LIN {X 0,Y 523.923,Z 138.219,A -85,B 0,C 180,E1 -4837.939,E2 -4837.939} C_VEL
LIN {X 0,Y 523.904,Z 138.224,A -85,B 0,C 180,E1 -4840.405,E2 -4840.405} C_VEL
LIN {X 0,Y 523.904,Z 138.223,A -85,B 0,C 180,E1 -4842.835,E2 -4842.835} C_VEL
LIN {X 0,Y 523.924,Z 138.217,A -85,B 0,C 180,E1 -4845.234,E2 -4845.234} C_VEL
LIN {X 0,Y 523.964,Z 138.218,A -85,B 0,C 180,E1 -4848.393,E2 -4848.393} C_VEL
LIN {X 0,Y 523.949,Z 138.215,A -85,B 0,C 180,E1 -4851.515,E2 -4851.515} C_VEL
LIN {X 0,Y 524.03,Z 138.208,A -85,B 0,C 180,E1 -4854.613,E2 -4854.613} C_VEL
LIN {X 0,Y 524.106,Z 138.195,A -85,B 0,C 180,E1 -4857.694,E2 -4857.694} C_VEL
LIN {X 0,Y 524.1,Z 138.202,A -85,B 0,C 180,E1 -4860,E2 -4860} C_VEL
LIN {X 0,Y 524.107,Z 138.201,A -85,B 0,C 180,E1 -4862.306,E2 -4862.306} C_VEL
LIN {X 0,Y 524.004,Z 138.215,A -85,B 0,C 180,E1 -4866.16,E2 -4866.16} C_VEL
LIN {X 0,Y 523.948,Z 138.215,A -85,B 0,C 180,E1 -4869.263,E2 -4869.263} C_VEL
LIN {X 0,Y 523.949,Z 138.217,A -85,B 0,C 180,E1 -4872.393,E2 -4872.393} C_VEL
LIN {X 0,Y 523.916,Z 138.224,A -85,B 0,C 180,E1 -4875.562,E2 -4875.562} C_VEL
LIN {X 0,Y 523.916,Z 138.219,A -85,B 0,C 180,E1 -4878.781,E2 -4878.781} C_VEL
LIN {X 0,Y 523.907,Z 138.222,A -85,B 0,C 180,E1 -4881.235,E2 -4881.235} C_VEL
LIN {X 0,Y 523.936,Z 138.22,A -85,B 0,C 180,E1 -4884.196,E2 -4884.196} C_VEL
LIN {X 0,Y 523.9,Z 138.226,A -85,B 0,C 180,E1 -4887.136,E2 -4887.136} C_VEL
LIN {X 0,Y 523.886,Z 138.23,A -85,B 0,C 180,E1 -4889.76,E2 -4889.76} C_VEL
LIN {X 0,Y 523.934,Z 138.219,A -85,B 0,C 180,E1 -4892.45,E2 -4892.45} C_VEL
LIN {X 0,Y 523.917,Z 138.226,A -85,B 0,C 180,E1 -4895.227,E2 -4895.227} C_VEL
LIN {X 0,Y 523.991,Z 138.296,A -85,B 0,C 180,E1 -4897.62,E2 -4897.62} C_VEL
LIN {X 0,Y 524.607,Z 144.392,A -85,B 0,C 180,E1 -4898.768,E2 -4898.768} C_VEL
LIN {X 0,Y 524.385,Z 160.445,A -85,B 0,C 180,E1 -4901.685,E2 -4901.685} C_VEL
LIN {X 0,Y 524.325,Z 167.357,A -85,B 0,C 180,E1 -4902.909,E2 -4902.909} C_VEL
LIN {X 0,Y 525.972,Z 176.481,A -85,B 0,C 180,E1 -4903.087,E2 -4903.087} C_VEL
LIN {X 0,Y 525.921,Z 195.473,A -85,B 0,C 180,E1 -4903.35,E2 -4903.35} C_VEL
LIN {X 0,Y 525.202,Z 201.318,A -85,B 0,C 180,E1 -4903.41,E2 -4903.41} C_VEL
LIN {X 0,Y 519.539,Z 220.31,A -85,B 0,C 180,E1 -4903.516,E2 -4903.516} C_VEL
LIN {X 0,Y 518.88,Z 226.152,A -85,B 0,C 180,E1 -4903.58,E2 -4903.58} C_VEL
LIN {X 0,Y 518.615,Z 274.692,A -85,B 0,C 180,E1 -4904.279,E2 -4904.279} C_VEL
LIN {X 0,Y 518.446,Z 287.858,A -85,B 0,C 180,E1 -4904.627,E2 -4904.627} C_VEL
LIN {X 0,Y 518.237,Z 299.345,A -85,B 0,C 180,E1 -4905.071,E2 -4905.071} C_VEL
LIN {X 0,Y 517.963,Z 309.998,A -85,B 0,C 180,E1 -4905.614,E2 -4905.614} C_VEL
LIN {X 0,Y 517.659,Z 320.815,A -85,B 0,C 180,E1 -4906.314,E2 -4906.314} C_VEL
LIN {X 0,Y 517.334,Z 331.814,A -85,B 0,C 180,E1 -4907.214,E2 -4907.214} C_VEL
LIN {X 0,Y 517.079,Z 341.89,A -85,B 0,C 180,E1 -4908.241,E2 -4908.241} C_VEL
LIN {X 0,Y 516.84,Z 349.994,A -85,B 0,C 180,E1 -4909.254,E2 -4909.254} C_VEL
LIN {X 0,Y 516.698,Z 356.638,A -85,B 0,C 180,E1 -4910.261,E2 -4910.261} C_VEL
LIN {X 0,Y 516.521,Z 363.204,A -85,B 0,C 180,E1 -4911.487,E2 -4911.487} C_VEL
LIN {X 0,Y 516.4,Z 368.418,A -85,B 0,C 180,E1 -4912.726,E2 -4912.726} C_VEL
LIN {X 0,Y 516.269,Z 372.957,A -85,B 0,C 180,E1 -4914.171,E2 -4914.171} C_VEL
LIN {X 0,Y 516.228,Z 375.099,A -85,B 0,C 180,E1 -4915.124,E2 -4915.124} C_VEL
LIN {X 0,Y 516.183,Z 376.74,A -85,B 0,C 180,E1 -4916.154,E2 -4916.154} C_VEL
LIN {X 0,Y 516.182,Z 377.808,A -85,B 0,C 180,E1 -4917.582,E2 -4917.582} C_VEL
LIN {X 0,Y 516.208,Z 377.531,A -85,B 0,C 180,E1 -4919.062,E2 -4919.062} C_VEL
LIN {X 0,Y 516.245,Z 375.742,A -85,B 0,C 180,E1 -4920.608,E2 -4920.608} C_VEL
LIN {X 0,Y 516.255,Z 373.847,A -85,B 0,C 180,E1 -4921.545,E2 -4921.545} C_VEL
LIN {X 0,Y 516.352,Z 370.125,A -85,B 0,C 180,E1 -4922.873,E2 -4922.873} C_VEL
LIN {X 0,Y 516.487,Z 365.084,A -85,B 0,C 180,E1 -4924.187,E2 -4924.187} C_VEL
LIN {X 0,Y 516.59,Z 358.966,A -85,B 0,C 180,E1 -4925.416,E2 -4925.416} C_VEL
LIN {X 0,Y 516.767,Z 351.875,A -85,B 0,C 180,E1 -4926.559,E2 -4926.559} C_VEL
LIN {X 0,Y 517,Z 343.744,A -85,B 0,C 180,E1 -4927.627,E2 -4927.627} C_VEL
LIN {X 0,Y 517.281,Z 333.786,A -85,B 0,C 180,E1 -4928.688,E2 -4928.688} C_VEL
LIN {X 0,Y 517.613,Z 322.557,A -85,B 0,C 180,E1 -4929.639,E2 -4929.639} C_VEL
LIN {X 0,Y 517.953,Z 311.621,A -85,B 0,C 180,E1 -4930.377,E2 -4930.377} C_VEL
LIN {X 0,Y 518.172,Z 299.685,A -85,B 0,C 180,E1 -4931.003,E2 -4931.003} C_VEL
LIN {X 0,Y 518.477,Z 286.399,A -85,B 0,C 180,E1 -4931.509,E2 -4931.509} C_VEL
LIN {X 0,Y 518.628,Z 274.047,A -85,B 0,C 180,E1 -4931.824,E2 -4931.824} C_VEL
LIN {X 0,Y 519.033,Z 177.008,A -85,B 0,C 180,E1 -4933.201,E2 -4933.201} C_VEL
LIN {X 0,Y 517.288,Z 167.26,A -85,B 0,C 180,E1 -4933.397,E2 -4933.397} C_VEL
LIN {X 0,Y 517.567,Z 152.131,A -85,B 0,C 180,E1 -4936.253,E2 -4936.253} C_VEL
LIN {X 0,Y 517.652,Z 143.863,A -85,B 0,C 180,E1 -4937.83,E2 -4937.83} C_VEL
LIN {X 0,Y 516.982,Z 139.092,A -85,B 0,C 180,E1 -4938.78,E2 -4938.78} C_VEL
LIN {X 0,Y 516.956,Z 139.089,A -85,B 0,C 180,E1 -4941.399,E2 -4941.399} C_VEL
LIN {X 0,Y 517.014,Z 139.087,A -85,B 0,C 180,E1 -4944.54,E2 -4944.54} C_VEL
LIN {X 0,Y 517.082,Z 139.07,A -85,B 0,C 180,E1 -4947.663,E2 -4947.663} C_VEL
LIN {X 0,Y 517.09,Z 139.072,A -85,B 0,C 180,E1 -4950.779,E2 -4950.779} C_VEL
LIN {X 0,Y 516.949,Z 139.087,A -85,B 0,C 180,E1 -4953.117,E2 -4953.117} C_VEL
LIN {X 0,Y 516.975,Z 139.092,A -85,B 0,C 180,E1 -4956.244,E2 -4956.244} C_VEL
LIN {X 0,Y 516.94,Z 139.088,A -85,B 0,C 180,E1 -4959.39,E2 -4959.39} C_VEL
LIN {X 0,Y 516.956,Z 139.09,A -85,B 0,C 180,E1 -4961.807,E2 -4961.807} C_VEL
LIN {X 0,Y 516.942,Z 139.088,A -85,B 0,C 180,E1 -4965.144,E2 -4965.144} C_VEL
LIN {X 0,Y 516.878,Z 139.1,A -85,B 0,C 180,E1 -4968.224,E2 -4968.224} C_VEL
LIN {X 0,Y 516.902,Z 139.093,A -85,B 0,C 180,E1 -4970.702,E2 -4970.702} C_VEL
LIN {X 0,Y 516.859,Z 139.099,A -85,B 0,C 180,E1 -4973.224,E2 -4973.224} C_VEL
LIN {X 0,Y 516.884,Z 139.098,A -85,B 0,C 180,E1 -4976.182,E2 -4976.182} C_VEL
LIN {X 0,Y 516.906,Z 139.096,A -85,B 0,C 180,E1 -4979.306,E2 -4979.306} C_VEL
LIN {X 0,Y 516.897,Z 139.093,A -85,B 0,C 180,E1 -4982.543,E2 -4982.543} C_VEL
LIN {X 0,Y 516.863,Z 139.103,A -85,B 0,C 180,E1 -4985.329,E2 -4985.329} C_VEL
LIN {X 0,Y 516.88,Z 139.098,A -85,B 0,C 180,E1 -4987.943,E2 -4987.943} C_VEL
LIN {X 0,Y 516.856,Z 139.099,A -85,B 0,C 180,E1 -4990.745,E2 -4990.745} C_VEL
LIN {X 0,Y 516.883,Z 139.096,A -85,B 0,C 180,E1 -4993.904,E2 -4993.904} C_VEL
LIN {X 0,Y 516.883,Z 139.095,A -85,B 0,C 180,E1 -4996.107,E2 -4996.107} C_VEL
LIN {X 0,Y 516.856,Z 139.106,A -85,B 0,C 180,E1 -4999.255,E2 -4999.255} C_VEL
LIN {X 0,Y 516.863,Z 139.097,A -85,B 0,C 180,E1 -5002.274,E2 -5002.274} C_VEL
LIN {X 0,Y 516.876,Z 139.103,A -85,B 0,C 180,E1 -5005.174,E2 -5005.174} C_VEL
LIN {X 0,Y 516.869,Z 139.096,A -85,B 0,C 180,E1 -5007.975,E2 -5007.975} C_VEL
LIN {X 0,Y 516.902,Z 139.098,A -85,B 0,C 180,E1 -5010.694,E2 -5010.694} C_VEL
LIN {X 0,Y 516.885,Z 139.094,A -85,B 0,C 180,E1 -5013.818,E2 -5013.818} C_VEL
LIN {X 0,Y 516.847,Z 139.108,A -85,B 0,C 180,E1 -5016.775,E2 -5016.775} C_VEL
LIN {X 0,Y 516.911,Z 139.091,A -85,B 0,C 180,E1 -5019.742,E2 -5019.742} C_VEL
LIN {X 0,Y 516.869,Z 139.105,A -85,B 0,C 180,E1 -5022.594,E2 -5022.594} C_VEL
LIN {X 0,Y 516.935,Z 139.091,A -85,B 0,C 180,E1 -5025.03,E2 -5025.03} C_VEL
LIN {X 0,Y 516.972,Z 139.089,A -85,B 0,C 180,E1 -5028.234,E2 -5028.234} C_VEL
LIN {X 0,Y 516.925,Z 139.09,A -85,B 0,C 180,E1 -5031.399,E2 -5031.399} C_VEL
LIN {X 0,Y 516.984,Z 139.088,A -85,B 0,C 180,E1 -5034.539,E2 -5034.539} C_VEL
LIN {X 0,Y 517.076,Z 139.072,A -85,B 0,C 180,E1 -5037.663,E2 -5037.663} C_VEL
LIN {X 0,Y 517.069,Z 139.078,A -85,B 0,C 180,E1 -5040,E2 -5040} C_VEL
LIN {X 0,Y 517.076,Z 139.077,A -85,B 0,C 180,E1 -5042.337,E2 -5042.337} C_VEL
LIN {X 0,Y 516.971,Z 139.09,A -85,B 0,C 180,E1 -5046.244,E2 -5046.244} C_VEL
LIN {X 0,Y 516.91,Z 139.093,A -85,B 0,C 180,E1 -5049.39,E2 -5049.39} C_VEL
LIN {X 0,Y 516.89,Z 139.095,A -85,B 0,C 180,E1 -5052.565,E2 -5052.565} C_VEL
LIN {X 0,Y 516.888,Z 139.095,A -85,B 0,C 180,E1 -5055.121,E2 -5055.121} C_VEL
LIN {X 0,Y 516.85,Z 139.101,A -85,B 0,C 180,E1 -5058.225,E2 -5058.225} C_VEL
LIN {X 0,Y 516.866,Z 139.097,A -85,B 0,C 180,E1 -5060.703,E2 -5060.703} C_VEL
LIN {X 0,Y 516.843,Z 139.103,A -85,B 0,C 180,E1 -5063.225,E2 -5063.225} C_VEL
LIN {X 0,Y 516.864,Z 139.098,A -85,B 0,C 180,E1 -5066.177,E2 -5066.177} C_VEL
LIN {X 0,Y 516.832,Z 139.101,A -85,B 0,C 180,E1 -5068.421,E2 -5068.421} C_VEL
LIN {X 0,Y 516.851,Z 139.103,A -85,B 0,C 180,E1 -5071.112,E2 -5071.112} C_VEL
LIN {X 0,Y 516.871,Z 139.098,A -85,B 0,C 180,E1 -5073.959,E2 -5073.959} C_VEL
LIN {X 0,Y 516.809,Z 139.106,A -85,B 0,C 180,E1 -5076.752,E2 -5076.752} C_VEL
LIN {X 0,Y 516.856,Z 139.1,A -85,B 0,C 180,E1 -5079.724,E2 -5079.724} C_VEL
LIN {X 0,Y 516.843,Z 139.104,A -85,B 0,C 180,E1 -5082.836,E2 -5082.836} C_VEL
LIN {X 0,Y 516.898,Z 139.101,A -85,B 0,C 180,E1 -5085.007,E2 -5085.007} C_VEL
LIN {X 0,Y 516.849,Z 139.1,A -85,B 0,C 180,E1 -5088.407,E2 -5088.407} C_VEL
LIN {X 0,Y 516.861,Z 139.102,A -85,B 0,C 180,E1 -5091.282,E2 -5091.282} C_VEL
LIN {X 0,Y 516.828,Z 139.108,A -85,B 0,C 180,E1 -5094.677,E2 -5094.677} C_VEL
LIN {X 0,Y 516.865,Z 139.098,A -85,B 0,C 180,E1 -5097.462,E2 -5097.462} C_VEL
LIN {X 0,Y 516.839,Z 139.108,A -85,B 0,C 180,E1 -5100.491,E2 -5100.491} C_VEL
LIN {X 0,Y 516.83,Z 139.106,A -85,B 0,C 180,E1 -5103.337,E2 -5103.337} C_VEL
LIN {X 0,Y 516.882,Z 139.297,A -85,B 0,C 180,E1 -5105.735,E2 -5105.735} C_VEL
LIN {X 0,Y 518.332,Z 147.82,A -85,B 0,C 180,E1 -5107.221,E2 -5107.221} C_VEL
LIN {X 0,Y 517.928,Z 164.685,A -85,B 0,C 180,E1 -5109.978,E2 -5109.978} C_VEL
LIN {X 0,Y 517.496,Z 182.348,A -85,B 0,C 180,E1 -5112.819,E2 -5112.819} C_VEL
LIN {X 0,Y 517.24,Z 193.77,A -85,B 0,C 180,E1 -5114.636,E2 -5114.636} C_VEL
LIN {X 0,Y 519.026,Z 206.371,A -85,B 0,C 180,E1 -5114.868,E2 -5114.868} C_VEL
LIN {X 0,Y 518.573,Z 302.296,A -85,B 0,C 180,E1 -5116.23,E2 -5116.23} C_VEL
LIN {X 0,Y 518.333,Z 316.173,A -85,B 0,C 180,E1 -5116.598,E2 -5116.598} C_VEL
LIN {X 0,Y 518.051,Z 329.122,A -85,B 0,C 180,E1 -5117.115,E2 -5117.115} C_VEL
LIN {X 0,Y 517.733,Z 341.445,A -85,B 0,C 180,E1 -5117.788,E2 -5117.788} C_VEL
LIN {X 0,Y 517.469,Z 352.266,A -85,B 0,C 180,E1 -5118.543,E2 -5118.543} C_VEL
LIN {X 0,Y 517.166,Z 362.51,A -85,B 0,C 180,E1 -5119.429,E2 -5119.429} C_VEL
LIN {X 0,Y 516.902,Z 371.715,A -85,B 0,C 180,E1 -5120.412,E2 -5120.412} C_VEL
LIN {X 0,Y 516.652,Z 380.678,A -85,B 0,C 180,E1 -5121.591,E2 -5121.591} C_VEL
LIN {X 0,Y 516.502,Z 387.894,A -85,B 0,C 180,E1 -5122.769,E2 -5122.769} C_VEL
LIN {X 0,Y 516.404,Z 394.464,A -85,B 0,C 180,E1 -5124.142,E2 -5124.142} C_VEL
LIN {X 0,Y 516.267,Z 398.806,A -85,B 0,C 180,E1 -5125.315,E2 -5125.315} C_VEL
LIN {X 0,Y 516.352,Z 401.108,A -85,B 0,C 180,E1 -5126.098,E2 -5126.098} C_VEL
LIN {X 0,Y 516.282,Z 402.97,A -85,B 0,C 180,E1 -5126.879,E2 -5126.879} C_VEL
LIN {X 0,Y 516.261,Z 404.367,A -85,B 0,C 180,E1 -5127.659,E2 -5127.659} C_VEL
LIN {X 0,Y 516.162,Z 405.968,A -85,B 0,C 180,E1 -5129.22,E2 -5129.22} C_VEL
LIN {X 0,Y 516.159,Z 406.183,A -85,B 0,C 180,E1 -5130,E2 -5130} C_VEL
LIN {X 0,Y 516.192,Z 405.356,A -85,B 0,C 180,E1 -5131.56,E2 -5131.56} C_VEL
LIN {X 0,Y 516.261,Z 404.358,A -85,B 0,C 180,E1 -5132.341,E2 -5132.341} C_VEL
LIN {X 0,Y 516.282,Z 402.958,A -85,B 0,C 180,E1 -5133.121,E2 -5133.121} C_VEL
LIN {X 0,Y 516.31,Z 400.014,A -85,B 0,C 180,E1 -5134.294,E2 -5134.294} C_VEL
LIN {X 0,Y 516.368,Z 396.03,A -85,B 0,C 180,E1 -5135.467,E2 -5135.467} C_VEL
LIN {X 0,Y 516.441,Z 390.135,A -85,B 0,C 180,E1 -5136.793,E2 -5136.793} C_VEL
LIN {X 0,Y 516.586,Z 383.2,A -85,B 0,C 180,E1 -5138.016,E2 -5138.016} C_VEL
LIN {X 0,Y 516.801,Z 374.888,A -85,B 0,C 180,E1 -5139.195,E2 -5139.195} C_VEL
LIN {X 0,Y 517.005,Z 366.359,A -85,B 0,C 180,E1 -5140.179,E2 -5140.179} C_VEL
LIN {X 0,Y 517.337,Z 355.824,A -85,B 0,C 180,E1 -5141.162,E2 -5141.162} C_VEL
LIN {X 0,Y 517.648,Z 344.821,A -85,B 0,C 180,E1 -5141.989,E2 -5141.989} C_VEL
LIN {X 0,Y 517.935,Z 333.952,A -85,B 0,C 180,E1 -5142.639,E2 -5142.639} C_VEL
LIN {X 0,Y 518.204,Z 322.146,A -85,B 0,C 180,E1 -5143.18,E2 -5143.18} C_VEL
LIN {X 0,Y 518.486,Z 308.535,A -85,B 0,C 180,E1 -5143.622,E2 -5143.622} C_VEL
LIN {X 0,Y 518.664,Z 296.421,A -85,B 0,C 180,E1 -5143.867,E2 -5143.867} C_VEL
LIN {X 0,Y 518.974,Z 204.763,A -85,B 0,C 180,E1 -5145.154,E2 -5145.154} C_VEL
LIN {X 0,Y 517.226,Z 193.408,A -85,B 0,C 180,E1 -5145.389,E2 -5145.389} C_VEL
LIN {X 0,Y 517.683,Z 174.421,A -85,B 0,C 180,E1 -5148.4,E2 -5148.4} C_VEL
LIN {X 0,Y 518.12,Z 155.212,A -85,B 0,C 180,E1 -5151.484,E2 -5151.484} C_VEL
LIN {X 0,Y 518.214,Z 146.498,A -85,B 0,C 180,E1 -5152.904,E2 -5152.904} C_VEL
LIN {X 0,Y 516.884,Z 139.1,A -85,B 0,C 180,E1 -5154.217,E2 -5154.217} C_VEL
LIN {X 0,Y 516.868,Z 139.106,A -85,B 0,C 180,E1 -5157.536,E2 -5157.536} C_VEL
LIN {X 0,Y 516.837,Z 139.104,A -85,B 0,C 180,E1 -5160.208,E2 -5160.208} C_VEL
LIN {X 0,Y 516.86,Z 139.106,A -85,B 0,C 180,E1 -5162.95,E2 -5162.95} C_VEL
LIN {X 0,Y 516.803,Z 139.107,A -85,B 0,C 180,E1 -5165.786,E2 -5165.786} C_VEL
LIN {X 0,Y 516.854,Z 139.103,A -85,B 0,C 180,E1 -5168.719,E2 -5168.719} C_VEL
LIN {X 0,Y 516.832,Z 139.103,A -85,B 0,C 180,E1 -5171.784,E2 -5171.784} C_VEL
LIN {X 0,Y 516.899,Z 139.101,A -85,B 0,C 180,E1 -5175.007,E2 -5175.007} C_VEL
LIN {X 0,Y 516.832,Z 139.104,A -85,B 0,C 180,E1 -5178.41,E2 -5178.41} C_VEL
LIN {X 0,Y 516.856,Z 139.103,A -85,B 0,C 180,E1 -5181.282,E2 -5181.282} C_VEL
LIN {X 0,Y 516.827,Z 139.108,A -85,B 0,C 180,E1 -5184.677,E2 -5184.677} C_VEL
LIN {X 0,Y 516.866,Z 139.097,A -85,B 0,C 180,E1 -5187.463,E2 -5187.463} C_VEL
LIN {X 0,Y 516.841,Z 139.105,A -85,B 0,C 180,E1 -5190.491,E2 -5190.491} C_VEL
LIN {X 0,Y 516.831,Z 139.102,A -85,B 0,C 180,E1 -5193.337,E2 -5193.337} C_VEL
LIN {X 0,Y 516.861,Z 139.096,A -85,B 0,C 180,E1 -5195.925,E2 -5195.925} C_VEL
LIN {X 0,Y 516.853,Z 139.106,A -85,B 0,C 180,E1 -5198.461,E2 -5198.461} C_VEL
LIN {X 0,Y 516.849,Z 139.103,A -85,B 0,C 180,E1 -5200.953,E2 -5200.953} C_VEL
LIN {X 0,Y 516.836,Z 139.099,A -85,B 0,C 180,E1 -5203.408,E2 -5203.408} C_VEL
LIN {X 0,Y 516.852,Z 139.1,A -85,B 0,C 180,E1 -5205.832,E2 -5205.832} C_VEL
LIN {X 0,Y 516.924,Z 139.096,A -85,B 0,C 180,E1 -5208.233,E2 -5208.233} C_VEL
LIN {X 0,Y 516.923,Z 139.09,A -85,B 0,C 180,E1 -5211.399,E2 -5211.399} C_VEL
LIN {X 0,Y 516.981,Z 139.087,A -85,B 0,C 180,E1 -5214.539,E2 -5214.539} C_VEL
LIN {X 0,Y 517.075,Z 139.071,A -85,B 0,C 180,E1 -5217.663,E2 -5217.663} C_VEL
LIN {X 0,Y 517.069,Z 139.078,A -85,B 0,C 180,E1 -5220,E2 -5220} C_VEL
LIN {X 0,Y 517.076,Z 139.076,A -85,B 0,C 180,E1 -5222.337,E2 -5222.337} C_VEL
LIN {X 0,Y 516.971,Z 139.09,A -85,B 0,C 180,E1 -5226.244,E2 -5226.244} C_VEL
LIN {X 0,Y 516.91,Z 139.092,A -85,B 0,C 180,E1 -5229.39,E2 -5229.39} C_VEL
LIN {X 0,Y 516.902,Z 139.093,A -85,B 0,C 180,E1 -5232.565,E2 -5232.565} C_VEL
LIN {X 0,Y 516.941,Z 139.089,A -85,B 0,C 180,E1 -5235.142,E2 -5235.142} C_VEL
LIN {X 0,Y 516.873,Z 139.1,A -85,B 0,C 180,E1 -5238.224,E2 -5238.224} C_VEL
LIN {X 0,Y 516.875,Z 139.096,A -85,B 0,C 180,E1 -5240.703,E2 -5240.703} C_VEL
LIN {X 0,Y 516.846,Z 139.103,A -85,B 0,C 180,E1 -5243.225,E2 -5243.225} C_VEL
LIN {X 0,Y 516.883,Z 139.099,A -85,B 0,C 180,E1 -5246.181,E2 -5246.181} C_VEL
LIN {X 0,Y 516.894,Z 139.101,A -85,B 0,C 180,E1 -5249.306,E2 -5249.306} C_VEL
LIN {X 0,Y 516.896,Z 139.096,A -85,B 0,C 180,E1 -5252.542,E2 -5252.542} C_VEL
LIN {X 0,Y 516.864,Z 139.106,A -85,B 0,C 180,E1 -5255.328,E2 -5255.328} C_VEL
LIN {X 0,Y 516.919,Z 139.106,A -85,B 0,C 180,E1 -5257.475,E2 -5257.475} C_VEL
LIN {X 0,Y 517.609,Z 144.246,A -85,B 0,C 180,E1 -5258.46,E2 -5258.46} C_VEL
LIN {X 0,Y 517.433,Z 158.995,A -85,B 0,C 180,E1 -5261.17,E2 -5261.17} C_VEL
LIN {X 0,Y 517.294,Z 167.36,A -85,B 0,C 180,E1 -5262.696,E2 -5262.696} C_VEL
LIN {X 0,Y 519.147,Z 177.868,A -85,B 0,C 180,E1 -5262.902,E2 -5262.902} C_VEL
LIN {X 0,Y 518.88,Z 226.152,A -85,B 0,C 180,E1 -5263.58,E2 -5263.58} C_VEL
LIN {X 0,Y 518.205,Z 231.997,A -85,B 0,C 180,E1 -5263.643,E2 -5263.643} C_VEL
LIN {X 0,Y 512.511,Z 250.987,A -85,B 0,C 180,E1 -5263.75,E2 -5263.75} C_VEL
LIN {X 0,Y 511.88,Z 256.829,A -85,B 0,C 180,E1 -5263.816,E2 -5263.816} C_VEL
LIN {X 0,Y 511.741,Z 276.642,A -85,B 0,C 180,E1 -5264.132,E2 -5264.132} C_VEL
LIN {X 0,Y 511.526,Z 289.245,A -85,B 0,C 180,E1 -5264.484,E2 -5264.484} C_VEL
LIN {X 0,Y 511.276,Z 301.879,A -85,B 0,C 180,E1 -5265.003,E2 -5265.003} C_VEL
LIN {X 0,Y 510.929,Z 313.813,A -85,B 0,C 180,E1 -5265.666,E2 -5265.666} C_VEL
LIN {X 0,Y 510.649,Z 323.936,A -85,B 0,C 180,E1 -5266.38,E2 -5266.38} C_VEL
LIN {X 0,Y 510.331,Z 334.534,A -85,B 0,C 180,E1 -5267.304,E2 -5267.304} C_VEL
LIN {X 0,Y 510.006,Z 343.981,A -85,B 0,C 180,E1 -5268.331,E2 -5268.331} C_VEL
LIN {X 0,Y 509.768,Z 352.414,A -85,B 0,C 180,E1 -5269.459,E2 -5269.459} C_VEL
LIN {X 0,Y 509.529,Z 359.455,A -85,B 0,C 180,E1 -5270.618,E2 -5270.618} C_VEL
LIN {X 0,Y 509.381,Z 365.472,A -85,B 0,C 180,E1 -5271.854,E2 -5271.854} C_VEL
LIN {X 0,Y 509.303,Z 370.387,A -85,B 0,C 180,E1 -5273.164,E2 -5273.164} C_VEL
LIN {X 0,Y 509.141,Z 374.221,A -85,B 0,C 180,E1 -5274.566,E2 -5274.566} C_VEL
LIN {X 0,Y 509.086,Z 376.655,A -85,B 0,C 180,E1 -5275.926,E2 -5275.926} C_VEL
LIN {X 0,Y 509.093,Z 377.969,A -85,B 0,C 180,E1 -5277.425,E2 -5277.425} C_VEL
LIN {X 0,Y 509.118,Z 377.859,A -85,B 0,C 180,E1 -5278.856,E2 -5278.856} C_VEL
LIN {X 0,Y 509.132,Z 376.278,A -85,B 0,C 180,E1 -5280.418,E2 -5280.418} C_VEL
LIN {X 0,Y 509.185,Z 374.104,A -85,B 0,C 180,E1 -5281.563,E2 -5281.563} C_VEL
LIN {X 0,Y 509.273,Z 370.409,A -85,B 0,C 180,E1 -5282.909,E2 -5282.909} C_VEL
LIN {X 0,Y 509.426,Z 365.403,A -85,B 0,C 180,E1 -5284.242,E2 -5284.242} C_VEL
LIN {X 0,Y 509.557,Z 358.926,A -85,B 0,C 180,E1 -5285.558,E2 -5285.558} C_VEL
LIN {X 0,Y 509.756,Z 350.795,A -85,B 0,C 180,E1 -5286.863,E2 -5286.863} C_VEL
LIN {X 0,Y 510.022,Z 342.281,A -85,B 0,C 180,E1 -5287.955,E2 -5287.955} C_VEL
LIN {X 0,Y 510.363,Z 331.972,A -85,B 0,C 180,E1 -5289.02,E2 -5289.02} C_VEL
LIN {X 0,Y 510.672,Z 321.732,A -85,B 0,C 180,E1 -5289.876,E2 -5289.876} C_VEL
LIN {X 0,Y 511.075,Z 310.445,A -85,B 0,C 180,E1 -5290.625,E2 -5290.625} C_VEL
LIN {X 0,Y 511.3,Z 297.836,A -85,B 0,C 180,E1 -5291.269,E2 -5291.269} C_VEL
LIN {X 0,Y 511.575,Z 285.248,A -85,B 0,C 180,E1 -5291.736,E2 -5291.736} C_VEL
LIN {X 0,Y 511.765,Z 271.826,A -85,B 0,C 180,E1 -5292.053,E2 -5292.053} C_VEL
LIN {X 0,Y 512.157,Z 177.465,A -85,B 0,C 180,E1 -5293.405,E2 -5293.405} C_VEL
LIN {X 0,Y 510.291,Z 167.361,A -85,B 0,C 180,E1 -5293.626,E2 -5293.626} C_VEL
LIN {X 0,Y 510.646,Z 151.393,A -85,B 0,C 180,E1 -5296.672,E2 -5296.672} C_VEL
LIN {X 0,Y 510.609,Z 144.09,A -85,B 0,C 180,E1 -5298.085,E2 -5298.085} C_VEL
LIN {X 0,Y 509.94,Z 139.968,A -85,B 0,C 180,E1 -5298.925,E2 -5298.925} C_VEL
LIN {X 0,Y 509.911,Z 139.969,A -85,B 0,C 180,E1 -5302.078,E2 -5302.078} C_VEL
LIN {X 0,Y 509.965,Z 139.965,A -85,B 0,C 180,E1 -5304.464,E2 -5304.464} C_VEL
LIN {X 0,Y 510.052,Z 139.946,A -85,B 0,C 180,E1 -5307.631,E2 -5307.631} C_VEL
LIN {X 0,Y 510.04,Z 139.95,A -85,B 0,C 180,E1 -5310.79,E2 -5310.79} C_VEL
LIN {X 0,Y 510.047,Z 139.955,A -85,B 0,C 180,E1 -5312.369,E2 -5312.369} C_VEL
LIN {X 0,Y 509.945,Z 139.96,A -85,B 0,C 180,E1 -5315.536,E2 -5315.536} C_VEL
LIN {X 0,Y 509.891,Z 139.968,A -85,B 0,C 180,E1 -5318.721,E2 -5318.721} C_VEL
LIN {X 0,Y 509.908,Z 139.97,A -85,B 0,C 180,E1 -5321.932,E2 -5321.932} C_VEL
LIN {X 0,Y 509.898,Z 139.965,A -85,B 0,C 180,E1 -5325.242,E2 -5325.242} C_VEL
LIN {X 0,Y 509.837,Z 139.974,A -85,B 0,C 180,E1 -5328.485,E2 -5328.485} C_VEL
LIN {X 0,Y 509.845,Z 139.972,A -85,B 0,C 180,E1 -5331.002,E2 -5331.002} C_VEL
LIN {X 0,Y 509.821,Z 139.98,A -85,B 0,C 180,E1 -5333.564,E2 -5333.564} C_VEL
LIN {X 0,Y 509.821,Z 139.976,A -85,B 0,C 180,E1 -5336.357,E2 -5336.357} C_VEL
LIN {X 0,Y 509.839,Z 139.972,A -85,B 0,C 180,E1 -5338.847,E2 -5338.847} C_VEL
LIN {X 0,Y 509.822,Z 139.983,A -85,B 0,C 180,E1 -5341.59,E2 -5341.59} C_VEL
LIN {X 0,Y 509.837,Z 139.973,A -85,B 0,C 180,E1 -5344.415,E2 -5344.415} C_VEL
LIN {X 0,Y 509.81,Z 139.983,A -85,B 0,C 180,E1 -5347.342,E2 -5347.342} C_VEL
LIN {X 0,Y 509.817,Z 139.975,A -85,B 0,C 180,E1 -5350.385,E2 -5350.385} C_VEL
LIN {X 0,Y 509.809,Z 139.981,A -85,B 0,C 180,E1 -5353.573,E2 -5353.573} C_VEL
LIN {X 0,Y 509.808,Z 139.976,A -85,B 0,C 180,E1 -5356.427,E2 -5356.427} C_VEL
LIN {X 0,Y 509.817,Z 139.978,A -85,B 0,C 180,E1 -5359.615,E2 -5359.615} C_VEL
LIN {X 0,Y 509.811,Z 139.979,A -85,B 0,C 180,E1 -5362.658,E2 -5362.658} C_VEL
LIN {X 0,Y 509.843,Z 139.972,A -85,B 0,C 180,E1 -5365.801,E2 -5365.801} C_VEL
LIN {X 0,Y 509.84,Z 139.978,A -85,B 0,C 180,E1 -5368.722,E2 -5368.722} C_VEL
LIN {X 0,Y 509.82,Z 139.975,A -85,B 0,C 180,E1 -5371.917,E2 -5371.917} C_VEL
LIN {X 0,Y 509.805,Z 139.984,A -85,B 0,C 180,E1 -5374.7,E2 -5374.7} C_VEL
LIN {X 0,Y 509.828,Z 139.974,A -85,B 0,C 180,E1 -5377.459,E2 -5377.459} C_VEL
LIN {X 0,Y 509.894,Z 139.966,A -85,B 0,C 180,E1 -5379.844,E2 -5379.844} C_VEL
LIN {X 0,Y 509.851,Z 139.976,A -85,B 0,C 180,E1 -5382.347,E2 -5382.347} C_VEL
LIN {X 0,Y 509.889,Z 139.971,A -85,B 0,C 180,E1 -5384.818,E2 -5384.818} C_VEL
LIN {X 0,Y 509.906,Z 139.968,A -85,B 0,C 180,E1 -5388.124,E2 -5388.124} C_VEL
LIN {X 0,Y 509.878,Z 139.968,A -85,B 0,C 180,E1 -5391.279,E2 -5391.279} C_VEL
LIN {X 0,Y 509.92,Z 139.963,A -85,B 0,C 180,E1 -5393.67,E2 -5393.67} C_VEL
LIN {X 0,Y 509.89,Z 139.968,A -85,B 0,C 180,E1 -5396.839,E2 -5396.839} C_VEL
LIN {X 0,Y 509.928,Z 139.967,A -85,B 0,C 180,E1 -5398.42,E2 -5398.42} C_VEL
LIN {X 0,Y 510.038,Z 139.954,A -85,B 0,C 180,E1 -5400,E2 -5400} C_VEL
LIN {X 0,Y 510.045,Z 139.952,A -85,B 0,C 180,E1 -5402.369,E2 -5402.369} C_VEL
LIN {X 0,Y 509.938,Z 139.962,A -85,B 0,C 180,E1 -5405.536,E2 -5405.536} C_VEL
LIN {X 0,Y 509.879,Z 139.975,A -85,B 0,C 180,E1 -5407.923,E2 -5407.923} C_VEL
LIN {X 0,Y 509.865,Z 139.969,A -85,B 0,C 180,E1 -5411.127,E2 -5411.127} C_VEL
LIN {X 0,Y 509.821,Z 139.979,A -85,B 0,C 180,E1 -5413.553,E2 -5413.553} C_VEL
LIN {X 0,Y 509.794,Z 139.984,A -85,B 0,C 180,E1 -5416.005,E2 -5416.005} C_VEL
LIN {X 0,Y 509.812,Z 139.976,A -85,B 0,C 180,E1 -5418.486,E2 -5418.486} C_VEL
LIN {X 0,Y 509.816,Z 139.976,A -85,B 0,C 180,E1 -5421.003,E2 -5421.003} C_VEL
LIN {X 0,Y 509.805,Z 139.985,A -85,B 0,C 180,E1 -5423.565,E2 -5423.565} C_VEL
LIN {X 0,Y 509.804,Z 139.977,A -85,B 0,C 180,E1 -5426.353,E2 -5426.353} C_VEL
LIN {X 0,Y 509.796,Z 139.979,A -85,B 0,C 180,E1 -5428.849,E2 -5428.849} C_VEL
LIN {X 0,Y 509.791,Z 139.985,A -85,B 0,C 180,E1 -5431.592,E2 -5431.592} C_VEL
LIN {X 0,Y 509.83,Z 139.973,A -85,B 0,C 180,E1 -5434.415,E2 -5434.415} C_VEL
LIN {X 0,Y 509.777,Z 139.988,A -85,B 0,C 180,E1 -5437.344,E2 -5437.344} C_VEL
LIN {X 0,Y 509.814,Z 139.976,A -85,B 0,C 180,E1 -5440.385,E2 -5440.385} C_VEL
LIN {X 0,Y 509.794,Z 139.981,A -85,B 0,C 180,E1 -5443.575,E2 -5443.575} C_VEL
LIN {X 0,Y 509.794,Z 139.979,A -85,B 0,C 180,E1 -5446.425,E2 -5446.425} C_VEL
LIN {X 0,Y 509.796,Z 139.979,A -85,B 0,C 180,E1 -5449.613,E2 -5449.613} C_VEL
LIN {X 0,Y 509.776,Z 139.985,A -85,B 0,C 180,E1 -5452.655,E2 -5452.655} C_VEL
LIN {X 0,Y 509.829,Z 139.973,A -85,B 0,C 180,E1 -5455.802,E2 -5455.802} C_VEL
LIN {X 0,Y 509.816,Z 139.984,A -85,B 0,C 180,E1 -5458.726,E2 -5458.726} C_VEL
LIN {X 0,Y 509.823,Z 139.978,A -85,B 0,C 180,E1 -5462.05,E2 -5462.05} C_VEL
LIN {X 0,Y 509.784,Z 139.988,A -85,B 0,C 180,E1 -5464.699,E2 -5464.699} C_VEL
LIN {X 0,Y 509.828,Z 140.028,A -85,B 0,C 180,E1 -5465.533,E2 -5465.533} C_VEL
LIN {X 0,Y 511.376,Z 148.534,A -85,B 0,C 180,E1 -5467.044,E2 -5467.044} C_VEL
LIN {X 0,Y 511.01,Z 163.696,A -85,B 0,C 180,E1 -5469.561,E2 -5469.561} C_VEL
LIN {X 0,Y 510.592,Z 178.964,A -85,B 0,C 180,E1 -5472.057,E2 -5472.057} C_VEL
LIN {X 0,Y 510.261,Z 193.653,A -85,B 0,C 180,E1 -5474.422,E2 -5474.422} C_VEL
LIN {X 0,Y 512.181,Z 206.085,A -85,B 0,C 180,E1 -5474.66,E2 -5474.66} C_VEL
LIN {X 0,Y 511.69,Z 301.999,A -85,B 0,C 180,E1 -5476.041,E2 -5476.041} C_VEL
LIN {X 0,Y 511.456,Z 315.147,A -85,B 0,C 180,E1 -5476.39,E2 -5476.39} C_VEL
LIN {X 0,Y 511.132,Z 327.819,A -85,B 0,C 180,E1 -5476.887,E2 -5476.887} C_VEL
LIN {X 0,Y 510.823,Z 339.597,A -85,B 0,C 180,E1 -5477.517,E2 -5477.517} C_VEL
LIN {X 0,Y 510.524,Z 350.748,A -85,B 0,C 180,E1 -5478.284,E2 -5478.284} C_VEL
LIN {X 0,Y 510.213,Z 361.239,A -85,B 0,C 180,E1 -5479.183,E2 -5479.183} C_VEL
LIN {X 0,Y 509.898,Z 369.813,A -85,B 0,C 180,E1 -5480.079,E2 -5480.079} C_VEL
LIN {X 0,Y 509.661,Z 377.723,A -85,B 0,C 180,E1 -5481.075,E2 -5481.075} C_VEL
LIN {X 0,Y 509.461,Z 385.449,A -85,B 0,C 180,E1 -5482.27,E2 -5482.27} C_VEL
LIN {X 0,Y 509.308,Z 392.562,A -85,B 0,C 180,E1 -5483.662,E2 -5483.662} C_VEL
LIN {X 0,Y 509.241,Z 397.295,A -85,B 0,C 180,E1 -5484.853,E2 -5484.853} C_VEL
LIN {X 0,Y 509.245,Z 400.912,A -85,B 0,C 180,E1 -5486.043,E2 -5486.043} C_VEL
LIN {X 0,Y 509.2,Z 402.776,A -85,B 0,C 180,E1 -5486.835,E2 -5486.835} C_VEL
LIN {X 0,Y 509.19,Z 404.173,A -85,B 0,C 180,E1 -5487.627,E2 -5487.627} C_VEL
LIN {X 0,Y 509.076,Z 405.774,A -85,B 0,C 180,E1 -5489.209,E2 -5489.209} C_VEL
LIN {X 0,Y 509.07,Z 405.989,A -85,B 0,C 180,E1 -5490,E2 -5490} C_VEL
LIN {X 0,Y 509.112,Z 405.16,A -85,B 0,C 180,E1 -5491.582,E2 -5491.582} C_VEL
LIN {X 0,Y 509.19,Z 404.162,A -85,B 0,C 180,E1 -5492.373,E2 -5492.373} C_VEL
LIN {X 0,Y 509.2,Z 402.76,A -85,B 0,C 180,E1 -5493.165,E2 -5493.165} C_VEL
LIN {X 0,Y 509.202,Z 399.813,A -85,B 0,C 180,E1 -5494.354,E2 -5494.354} C_VEL
LIN {X 0,Y 509.284,Z 395.825,A -85,B 0,C 180,E1 -5495.543,E2 -5495.543} C_VEL
LIN {X 0,Y 509.395,Z 389.792,A -85,B 0,C 180,E1 -5496.914,E2 -5496.914} C_VEL
LIN {X 0,Y 509.536,Z 382.986,A -85,B 0,C 180,E1 -5498.128,E2 -5498.128} C_VEL
LIN {X 0,Y 509.745,Z 374.668,A -85,B 0,C 180,E1 -5499.323,E2 -5499.323} C_VEL
LIN {X 0,Y 509.978,Z 366.133,A -85,B 0,C 180,E1 -5500.321,E2 -5500.321} C_VEL
LIN {X 0,Y 510.351,Z 355.589,A -85,B 0,C 180,E1 -5501.317,E2 -5501.317} C_VEL
LIN {X 0,Y 510.652,Z 344.578,A -85,B 0,C 180,E1 -5502.156,E2 -5502.156} C_VEL
LIN {X 0,Y 510.987,Z 333.697,A -85,B 0,C 180,E1 -5502.814,E2 -5502.814} C_VEL
LIN {X 0,Y 511.269,Z 321.871,A -85,B 0,C 180,E1 -5503.362,E2 -5503.362} C_VEL
LIN {X 0,Y 511.572,Z 308.237,A -85,B 0,C 180,E1 -5503.81,E2 -5503.81} C_VEL
LIN {X 0,Y 511.788,Z 296.073,A -85,B 0,C 180,E1 -5504.057,E2 -5504.057} C_VEL
LIN {X 0,Y 512.096,Z 205.338,A -85,B 0,C 180,E1 -5505.351,E2 -5505.351} C_VEL
LIN {X 0,Y 510.218,Z 193.322,A -85,B 0,C 180,E1 -5505.587,E2 -5505.587} C_VEL
LIN {X 0,Y 510.722,Z 174.204,A -85,B 0,C 180,E1 -5508.66,E2 -5508.66} C_VEL
LIN {X 0,Y 511.167,Z 156.276,A -85,B 0,C 180,E1 -5511.579,E2 -5511.579} C_VEL
LIN {X 0,Y 511.304,Z 148.058,A -85,B 0,C 180,E1 -5512.937,E2 -5512.937} C_VEL
LIN {X 0,Y 509.822,Z 139.98,A -85,B 0,C 180,E1 -5514.374,E2 -5514.374} C_VEL
LIN {X 0,Y 509.815,Z 139.983,A -85,B 0,C 180,E1 -5517.06,E2 -5517.06} C_VEL
LIN {X 0,Y 509.785,Z 139.986,A -85,B 0,C 180,E1 -5519.756,E2 -5519.756} C_VEL
LIN {X 0,Y 509.822,Z 139.98,A -85,B 0,C 180,E1 -5522.765,E2 -5522.765} C_VEL
LIN {X 0,Y 509.778,Z 139.985,A -85,B 0,C 180,E1 -5525.571,E2 -5525.571} C_VEL
LIN {X 0,Y 509.801,Z 139.978,A -85,B 0,C 180,E1 -5528.343,E2 -5528.343} C_VEL
LIN {X 0,Y 509.784,Z 139.984,A -85,B 0,C 180,E1 -5531.433,E2 -5531.433} C_VEL
LIN {X 0,Y 509.837,Z 139.978,A -85,B 0,C 180,E1 -5534.671,E2 -5534.671} C_VEL
LIN {X 0,Y 509.785,Z 139.982,A -85,B 0,C 180,E1 -5537.505,E2 -5537.505} C_VEL
LIN {X 0,Y 509.809,Z 139.98,A -85,B 0,C 180,E1 -5540.644,E2 -5540.644} C_VEL
LIN {X 0,Y 509.761,Z 139.982,A -85,B 0,C 180,E1 -5543.641,E2 -5543.641} C_VEL
LIN {X 0,Y 509.825,Z 139.979,A -85,B 0,C 180,E1 -5546.536,E2 -5546.536} C_VEL
LIN {X 0,Y 509.804,Z 139.978,A -85,B 0,C 180,E1 -5549.331,E2 -5549.331} C_VEL
LIN {X 0,Y 509.825,Z 139.974,A -85,B 0,C 180,E1 -5552.05,E2 -5552.05} C_VEL
LIN {X 0,Y 509.786,Z 139.983,A -85,B 0,C 180,E1 -5554.699,E2 -5554.699} C_VEL
LIN {X 0,Y 509.827,Z 139.974,A -85,B 0,C 180,E1 -5557.459,E2 -5557.459} C_VEL
LIN {X 0,Y 509.81,Z 139.983,A -85,B 0,C 180,E1 -5560.679,E2 -5560.679} C_VEL
LIN {X 0,Y 509.791,Z 139.978,A -85,B 0,C 180,E1 -5563.172,E2 -5563.172} C_VEL
LIN {X 0,Y 509.818,Z 139.975,A -85,B 0,C 180,E1 -5565.633,E2 -5565.633} C_VEL
LIN {X 0,Y 509.892,Z 139.971,A -85,B 0,C 180,E1 -5568.132,E2 -5568.132} C_VEL
LIN {X 0,Y 509.876,Z 139.968,A -85,B 0,C 180,E1 -5571.279,E2 -5571.279} C_VEL
LIN {X 0,Y 509.9,Z 139.962,A -85,B 0,C 180,E1 -5573.669,E2 -5573.669} C_VEL
LIN {X 0,Y 509.887,Z 139.965,A -85,B 0,C 180,E1 -5576.839,E2 -5576.839} C_VEL
LIN {X 0,Y 509.927,Z 139.966,A -85,B 0,C 180,E1 -5578.42,E2 -5578.42} C_VEL
LIN {X 0,Y 510.038,Z 139.954,A -85,B 0,C 180,E1 -5580,E2 -5580} C_VEL
LIN {X 0,Y 510.044,Z 139.951,A -85,B 0,C 180,E1 -5582.369,E2 -5582.369} C_VEL
LIN {X 0,Y 509.938,Z 139.962,A -85,B 0,C 180,E1 -5585.536,E2 -5585.536} C_VEL
LIN {X 0,Y 509.879,Z 139.976,A -85,B 0,C 180,E1 -5587.923,E2 -5587.923} C_VEL
LIN {X 0,Y 509.866,Z 139.97,A -85,B 0,C 180,E1 -5591.127,E2 -5591.127} C_VEL
LIN {X 0,Y 509.829,Z 139.977,A -85,B 0,C 180,E1 -5593.553,E2 -5593.553} C_VEL
LIN {X 0,Y 509.807,Z 139.984,A -85,B 0,C 180,E1 -5596.005,E2 -5596.005} C_VEL
LIN {X 0,Y 509.83,Z 139.975,A -85,B 0,C 180,E1 -5598.485,E2 -5598.485} C_VEL
LIN {X 0,Y 509.822,Z 139.976,A -85,B 0,C 180,E1 -5601.003,E2 -5601.003} C_VEL
LIN {X 0,Y 509.813,Z 139.984,A -85,B 0,C 180,E1 -5603.564,E2 -5603.564} C_VEL
LIN {X 0,Y 509.819,Z 139.978,A -85,B 0,C 180,E1 -5606.356,E2 -5606.356} C_VEL
LIN {X 0,Y 509.828,Z 139.977,A -85,B 0,C 180,E1 -5608.847,E2 -5608.847} C_VEL
LIN {X 0,Y 509.815,Z 139.984,A -85,B 0,C 180,E1 -5611.591,E2 -5611.591} C_VEL
LIN {X 0,Y 509.838,Z 139.976,A -85,B 0,C 180,E1 -5614.415,E2 -5614.415} C_VEL
LIN {X 0,Y 509.877,Z 140.003,A -85,B 0,C 180,E1 -5617.336,E2 -5617.336} C_VEL
LIN {X 0,Y 510.666,Z 146.148,A -85,B 0,C 180,E1 -5618.517,E2 -5618.517} C_VEL
LIN {X 0,Y 510.426,Z 161.483,A -85,B 0,C 180,E1 -5621.369,E2 -5621.369} C_VEL
LIN {X 0,Y 510.3,Z 167.478,A -85,B 0,C 180,E1 -5622.474,E2 -5622.474} C_VEL
LIN {X 0,Y 512.324,Z 178.979,A -85,B 0,C 180,E1 -5622.709,E2 -5622.709} C_VEL
LIN {X 0,Y 511.88,Z 256.829,A -85,B 0,C 180,E1 -5623.816,E2 -5623.816} C_VEL
LIN {X 0,Y 511.236,Z 262.68,A -85,B 0,C 180,E1 -5623.879,E2 -5623.879} C_VEL
LIN {X 0,Y 508.347,Z 272.168,A -85,B 0,C 180,E1 -5623.945,E2 -5623.945} C_VEL
LIN {X 0,Y 505.398,Z 281.561,A -85,B 0,C 180,E1 -5624.07,E2 -5624.07} C_VEL
LIN {X 0,Y 504.654,Z 287.254,A -85,B 0,C 180,E1 -5624.223,E2 -5624.223} C_VEL
LIN {X 0,Y 504.417,Z 299.823,A -85,B 0,C 180,E1 -5624.717,E2 -5624.717} C_VEL
LIN {X 0,Y 504.088,Z 311.239,A -85,B 0,C 180,E1 -5625.32,E2 -5625.32} C_VEL
LIN {X 0,Y 503.737,Z 322.501,A -85,B 0,C 180,E1 -5626.09,E2 -5626.09} C_VEL
LIN {X 0,Y 503.342,Z 332.678,A -85,B 0,C 180,E1 -5626.958,E2 -5626.958} C_VEL
LIN {X 0,Y 503.059,Z 342.749,A -85,B 0,C 180,E1 -5628.022,E2 -5628.022} C_VEL
LIN {X 0,Y 502.768,Z 350.409,A -85,B 0,C 180,E1 -5629.012,E2 -5629.012} C_VEL
LIN {X 0,Y 502.554,Z 358.344,A -85,B 0,C 180,E1 -5630.278,E2 -5630.278} C_VEL
LIN {X 0,Y 502.337,Z 364.831,A -85,B 0,C 180,E1 -5631.58,E2 -5631.58} C_VEL
LIN {X 0,Y 502.234,Z 370.304,A -85,B 0,C 180,E1 -5633.006,E2 -5633.006} C_VEL
LIN {X 0,Y 502.086,Z 373.887,A -85,B 0,C 180,E1 -5634.278,E2 -5634.278} C_VEL
LIN {X 0,Y 502.022,Z 376.559,A -85,B 0,C 180,E1 -5635.687,E2 -5635.687} C_VEL
LIN {X 0,Y 501.975,Z 378.014,A -85,B 0,C 180,E1 -5637.145,E2 -5637.145} C_VEL
LIN {X 0,Y 502.005,Z 378.165,A -85,B 0,C 180,E1 -5638.649,E2 -5638.649} C_VEL
LIN {X 0,Y 502.026,Z 376.791,A -85,B 0,C 180,E1 -5640.222,E2 -5640.222} C_VEL
LIN {X 0,Y 502.101,Z 373.735,A -85,B 0,C 180,E1 -5641.864,E2 -5641.864} C_VEL
LIN {X 0,Y 502.185,Z 370.695,A -85,B 0,C 180,E1 -5642.946,E2 -5642.946} C_VEL
LIN {X 0,Y 502.346,Z 365.724,A -85,B 0,C 180,E1 -5644.297,E2 -5644.297} C_VEL
LIN {X 0,Y 502.435,Z 360.551,A -85,B 0,C 180,E1 -5645.397,E2 -5645.397} C_VEL
LIN {X 0,Y 502.641,Z 354.107,A -85,B 0,C 180,E1 -5646.516,E2 -5646.516} C_VEL
LIN {X 0,Y 502.939,Z 345.664,A -85,B 0,C 180,E1 -5647.7,E2 -5647.7} C_VEL
LIN {X 0,Y 503.238,Z 336.845,A -85,B 0,C 180,E1 -5648.709,E2 -5648.709} C_VEL
LIN {X 0,Y 503.58,Z 326.359,A -85,B 0,C 180,E1 -5649.686,E2 -5649.686} C_VEL
LIN {X 0,Y 503.934,Z 316.23,A -85,B 0,C 180,E1 -5650.445,E2 -5650.445} C_VEL
LIN {X 0,Y 504.255,Z 304.376,A -85,B 0,C 180,E1 -5651.145,E2 -5651.145} C_VEL
LIN {X 0,Y 504.533,Z 292.145,A -85,B 0,C 180,E1 -5651.691,E2 -5651.691} C_VEL
LIN {X 0,Y 504.775,Z 279.601,A -85,B 0,C 180,E1 -5652.086,E2 -5652.086} C_VEL
LIN {X 0,Y 504.927,Z 265.161,A -85,B 0,C 180,E1 -5652.352,E2 -5652.352} C_VEL
LIN {X 0,Y 505.338,Z 178.455,A -85,B 0,C 180,E1 -5653.604,E2 -5653.604} C_VEL
LIN {X 0,Y 503.321,Z 167.566,A -85,B 0,C 180,E1 -5653.838,E2 -5653.838} C_VEL
LIN {X 0,Y 503.734,Z 150.658,A -85,B 0,C 180,E1 -5657.101,E2 -5657.101} C_VEL
LIN {X 0,Y 503.498,Z 144.471,A -85,B 0,C 180,E1 -5658.323,E2 -5658.323} C_VEL
LIN {X 0,Y 502.9,Z 140.845,A -85,B 0,C 180,E1 -5659.074,E2 -5659.074} C_VEL
LIN {X 0,Y 502.875,Z 140.844,A -85,B 0,C 180,E1 -5661.966,E2 -5661.966} C_VEL
LIN {X 0,Y 502.919,Z 140.843,A -85,B 0,C 180,E1 -5664.386,E2 -5664.386} C_VEL
LIN {X 0,Y 503.02,Z 140.822,A -85,B 0,C 180,E1 -5667.598,E2 -5667.598} C_VEL
LIN {X 0,Y 502.992,Z 140.828,A -85,B 0,C 180,E1 -5670.801,E2 -5670.801} C_VEL
LIN {X 0,Y 503.014,Z 140.83,A -85,B 0,C 180,E1 -5672.402,E2 -5672.402} C_VEL
LIN {X 0,Y 502.901,Z 140.838,A -85,B 0,C 180,E1 -5675.614,E2 -5675.614} C_VEL
LIN {X 0,Y 502.854,Z 140.849,A -85,B 0,C 180,E1 -5678.034,E2 -5678.034} C_VEL
LIN {X 0,Y 502.879,Z 140.84,A -85,B 0,C 180,E1 -5681.283,E2 -5681.283} C_VEL
LIN {X 0,Y 502.834,Z 140.847,A -85,B 0,C 180,E1 -5684.571,E2 -5684.571} C_VEL
LIN {X 0,Y 502.812,Z 140.854,A -85,B 0,C 180,E1 -5688.109,E2 -5688.109} C_VEL
LIN {X 0,Y 502.833,Z 140.846,A -85,B 0,C 180,E1 -5690.536,E2 -5690.536} C_VEL
LIN {X 0,Y 502.789,Z 140.851,A -85,B 0,C 180,E1 -5693.041,E2 -5693.041} C_VEL
LIN {X 0,Y 502.781,Z 140.859,A -85,B 0,C 180,E1 -5695.679,E2 -5695.679} C_VEL
LIN {X 0,Y 502.775,Z 140.853,A -85,B 0,C 180,E1 -5698.377,E2 -5698.377} C_VEL
LIN {X 0,Y 502.795,Z 140.852,A -85,B 0,C 180,E1 -5701.144,E2 -5701.144} C_VEL
LIN {X 0,Y 502.789,Z 140.853,A -85,B 0,C 180,E1 -5703.995,E2 -5703.995} C_VEL
LIN {X 0,Y 502.767,Z 140.858,A -85,B 0,C 180,E1 -5707.176,E2 -5707.176} C_VEL
LIN {X 0,Y 502.775,Z 140.854,A -85,B 0,C 180,E1 -5710.017,E2 -5710.017} C_VEL
LIN {X 0,Y 502.75,Z 140.863,A -85,B 0,C 180,E1 -5713.234,E2 -5713.234} C_VEL
LIN {X 0,Y 502.781,Z 140.855,A -85,B 0,C 180,E1 -5715.66,E2 -5715.66} C_VEL
LIN {X 0,Y 502.768,Z 140.859,A -85,B 0,C 180,E1 -5719.012,E2 -5719.012} C_VEL
LIN {X 0,Y 502.793,Z 140.85,A -85,B 0,C 180,E1 -5722.046,E2 -5722.046} C_VEL
LIN {X 0,Y 502.795,Z 140.859,A -85,B 0,C 180,E1 -5725.034,E2 -5725.034} C_VEL
LIN {X 0,Y 502.781,Z 140.852,A -85,B 0,C 180,E1 -5727.915,E2 -5727.915} C_VEL
LIN {X 0,Y 502.794,Z 140.856,A -85,B 0,C 180,E1 -5730.71,E2 -5730.71} C_VEL
LIN {X 0,Y 502.778,Z 140.853,A -85,B 0,C 180,E1 -5733.46,E2 -5733.46} C_VEL
LIN {X 0,Y 502.765,Z 140.854,A -85,B 0,C 180,E1 -5736.085,E2 -5736.085} C_VEL
LIN {X 0,Y 502.834,Z 140.845,A -85,B 0,C 180,E1 -5739.464,E2 -5739.464} C_VEL
LIN {X 0,Y 502.789,Z 140.853,A -85,B 0,C 180,E1 -5742.09,E2 -5742.09} C_VEL
LIN {X 0,Y 502.826,Z 140.846,A -85,B 0,C 180,E1 -5745.429,E2 -5745.429} C_VEL
LIN {X 0,Y 502.88,Z 140.844,A -85,B 0,C 180,E1 -5748.717,E2 -5748.717} C_VEL
LIN {X 0,Y 502.851,Z 140.846,A -85,B 0,C 180,E1 -5751.966,E2 -5751.966} C_VEL
LIN {X 0,Y 502.896,Z 140.845,A -85,B 0,C 180,E1 -5754.386,E2 -5754.386} C_VEL
LIN {X 0,Y 503.012,Z 140.824,A -85,B 0,C 180,E1 -5757.598,E2 -5757.598} C_VEL
LIN {X 0,Y 503.007,Z 140.829,A -85,B 0,C 180,E1 -5760,E2 -5760} C_VEL
LIN {X 0,Y 503.012,Z 140.827,A -85,B 0,C 180,E1 -5762.402,E2 -5762.402} C_VEL
LIN {X 0,Y 502.895,Z 140.84,A -85,B 0,C 180,E1 -5765.614,E2 -5765.614} C_VEL
LIN {X 0,Y 502.85,Z 140.851,A -85,B 0,C 180,E1 -5768.034,E2 -5768.034} C_VEL
LIN {X 0,Y 502.841,Z 140.845,A -85,B 0,C 180,E1 -5771.284,E2 -5771.284} C_VEL
LIN {X 0,Y 502.802,Z 140.85,A -85,B 0,C 180,E1 -5774.572,E2 -5774.572} C_VEL
LIN {X 0,Y 502.782,Z 140.858,A -85,B 0,C 180,E1 -5777.91,E2 -5777.91} C_VEL
LIN {X 0,Y 502.772,Z 140.853,A -85,B 0,C 180,E1 -5780.517,E2 -5780.517} C_VEL
LIN {X 0,Y 502.783,Z 140.853,A -85,B 0,C 180,E1 -5783.041,E2 -5783.041} C_VEL
LIN {X 0,Y 502.765,Z 140.861,A -85,B 0,C 180,E1 -5785.68,E2 -5785.68} C_VEL
LIN {X 0,Y 502.762,Z 140.854,A -85,B 0,C 180,E1 -5788.378,E2 -5788.378} C_VEL
LIN {X 0,Y 502.768,Z 140.861,A -85,B 0,C 180,E1 -5791.493,E2 -5791.493} C_VEL
LIN {X 0,Y 502.782,Z 140.851,A -85,B 0,C 180,E1 -5794.44,E2 -5794.44} C_VEL
LIN {X 0,Y 502.731,Z 140.865,A -85,B 0,C 180,E1 -5797.17,E2 -5797.17} C_VEL
LIN {X 0,Y 502.751,Z 140.856,A -85,B 0,C 180,E1 -5800.019,E2 -5800.019} C_VEL
LIN {X 0,Y 502.747,Z 140.856,A -85,B 0,C 180,E1 -5802.192,E2 -5802.192} C_VEL
LIN {X 0,Y 502.78,Z 140.855,A -85,B 0,C 180,E1 -5805.471,E2 -5805.471} C_VEL
LIN {X 0,Y 502.76,Z 140.862,A -85,B 0,C 180,E1 -5808.928,E2 -5808.928} C_VEL
LIN {X 0,Y 502.755,Z 140.855,A -85,B 0,C 180,E1 -5812.042,E2 -5812.042} C_VEL
LIN {X 0,Y 502.769,Z 140.859,A -85,B 0,C 180,E1 -5815.031,E2 -5815.031} C_VEL
LIN {X 0,Y 502.757,Z 140.855,A -85,B 0,C 180,E1 -5817.913,E2 -5817.913} C_VEL
LIN {X 0,Y 502.753,Z 140.864,A -85,B 0,C 180,E1 -5820.707,E2 -5820.707} C_VEL
LIN {X 0,Y 502.771,Z 140.857,A -85,B 0,C 180,E1 -5823.461,E2 -5823.461} C_VEL
LIN {X 0,Y 502.794,Z 140.954,A -85,B 0,C 180,E1 -5825.362,E2 -5825.362} C_VEL
LIN {X 0,Y 504.434,Z 150.274,A -85,B 0,C 180,E1 -5827.039,E2 -5827.039} C_VEL
LIN {X 0,Y 504.005,Z 165.5,A -85,B 0,C 180,E1 -5829.598,E2 -5829.598} C_VEL
LIN {X 0,Y 503.575,Z 180.708,A -85,B 0,C 180,E1 -5832.119,E2 -5832.119} C_VEL
LIN {X 0,Y 503.257,Z 193.383,A -85,B 0,C 180,E1 -5834.199,E2 -5834.199} C_VEL
LIN {X 0,Y 505.319,Z 207.204,A -85,B 0,C 180,E1 -5834.467,E2 -5834.467} C_VEL
LIN {X 0,Y 504.804,Z 301.674,A -85,B 0,C 180,E1 -5835.847,E2 -5835.847} C_VEL
LIN {X 0,Y 504.569,Z 314.867,A -85,B 0,C 180,E1 -5836.2,E2 -5836.2} C_VEL
LIN {X 0,Y 504.201,Z 327.562,A -85,B 0,C 180,E1 -5836.703,E2 -5836.703} C_VEL
LIN {X 0,Y 503.89,Z 338.682,A -85,B 0,C 180,E1 -5837.299,E2 -5837.299} C_VEL
LIN {X 0,Y 503.54,Z 350.523,A -85,B 0,C 180,E1 -5838.12,E2 -5838.12} C_VEL
LIN {X 0,Y 503.221,Z 361.022,A -85,B 0,C 180,E1 -5839.03,E2 -5839.03} C_VEL
LIN {X 0,Y 502.849,Z 369.601,A -85,B 0,C 180,E1 -5839.938,E2 -5839.938} C_VEL
LIN {X 0,Y 502.619,Z 377.516,A -85,B 0,C 180,E1 -5840.949,E2 -5840.949} C_VEL
LIN {X 0,Y 502.384,Z 385.246,A -85,B 0,C 180,E1 -5842.161,E2 -5842.161} C_VEL
LIN {X 0,Y 502.235,Z 392.362,A -85,B 0,C 180,E1 -5843.572,E2 -5843.572} C_VEL
LIN {X 0,Y 502.172,Z 397.098,A -85,B 0,C 180,E1 -5844.781,E2 -5844.781} C_VEL
LIN {X 0,Y 502.137,Z 400.716,A -85,B 0,C 180,E1 -5845.987,E2 -5845.987} C_VEL
LIN {X 0,Y 502.12,Z 402.581,A -85,B 0,C 180,E1 -5846.791,E2 -5846.791} C_VEL
LIN {X 0,Y 502.092,Z 403.979,A -85,B 0,C 180,E1 -5847.593,E2 -5847.593} C_VEL
LIN {X 0,Y 501.992,Z 405.58,A -85,B 0,C 180,E1 -5849.198,E2 -5849.198} C_VEL
LIN {X 0,Y 501.984,Z 405.794,A -85,B 0,C 180,E1 -5850,E2 -5850} C_VEL
LIN {X 0,Y 502.036,Z 404.964,A -85,B 0,C 180,E1 -5851.604,E2 -5851.604} C_VEL
LIN {X 0,Y 502.092,Z 403.964,A -85,B 0,C 180,E1 -5852.407,E2 -5852.407} C_VEL
LIN {X 0,Y 502.12,Z 402.561,A -85,B 0,C 180,E1 -5853.21,E2 -5853.21} C_VEL
LIN {X 0,Y 502.1,Z 399.611,A -85,B 0,C 180,E1 -5854.415,E2 -5854.415} C_VEL
LIN {X 0,Y 502.199,Z 395.621,A -85,B 0,C 180,E1 -5855.622,E2 -5855.622} C_VEL
LIN {X 0,Y 502.327,Z 389.582,A -85,B 0,C 180,E1 -5857.012,E2 -5857.012} C_VEL
LIN {X 0,Y 502.47,Z 382.772,A -85,B 0,C 180,E1 -5858.243,E2 -5858.243} C_VEL
LIN {X 0,Y 502.711,Z 374.45,A -85,B 0,C 180,E1 -5859.455,E2 -5859.455} C_VEL
LIN {X 0,Y 502.966,Z 365.909,A -85,B 0,C 180,E1 -5860.466,E2 -5860.466} C_VEL
LIN {X 0,Y 503.362,Z 355.36,A -85,B 0,C 180,E1 -5861.476,E2 -5861.476} C_VEL
LIN {X 0,Y 503.694,Z 344.343,A -85,B 0,C 180,E1 -5862.327,E2 -5862.327} C_VEL
LIN {X 0,Y 504.03,Z 333.453,A -85,B 0,C 180,E1 -5862.994,E2 -5862.994} C_VEL
LIN {X 0,Y 504.335,Z 321.612,A -85,B 0,C 180,E1 -5863.55,E2 -5863.55} C_VEL
LIN {X 0,Y 504.666,Z 307.959,A -85,B 0,C 180,E1 -5864.003,E2 -5864.003} C_VEL
LIN {X 0,Y 504.92,Z 294.033,A -85,B 0,C 180,E1 -5864.278,E2 -5864.278} C_VEL
LIN {X 0,Y 505.216,Z 206.015,A -85,B 0,C 180,E1 -5865.553,E2 -5865.553} C_VEL
LIN {X 0,Y 503.211,Z 193.068,A -85,B 0,C 180,E1 -5865.818,E2 -5865.818} C_VEL
LIN {X 0,Y 503.739,Z 173.991,A -85,B 0,C 180,E1 -5868.928,E2 -5868.928} C_VEL
LIN {X 0,Y 504.219,Z 157.362,A -85,B 0,C 180,E1 -5871.677,E2 -5871.677} C_VEL
LIN {X 0,Y 504.276,Z 148.904,A -85,B 0,C 180,E1 -5873.098,E2 -5873.098} C_VEL
LIN {X 0,Y 502.766,Z 140.859,A -85,B 0,C 180,E1 -5874.536,E2 -5874.536} C_VEL
LIN {X 0,Y 502.77,Z 140.861,A -85,B 0,C 180,E1 -5877.471,E2 -5877.471} C_VEL
LIN {X 0,Y 502.744,Z 140.861,A -85,B 0,C 180,E1 -5880.216,E2 -5880.216} C_VEL
LIN {X 0,Y 502.769,Z 140.862,A -85,B 0,C 180,E1 -5883.036,E2 -5883.036} C_VEL
LIN {X 0,Y 502.737,Z 140.859,A -85,B 0,C 180,E1 -5885.955,E2 -5885.955} C_VEL
LIN {X 0,Y 502.765,Z 140.861,A -85,B 0,C 180,E1 -5888.98,E2 -5888.98} C_VEL
LIN {X 0,Y 502.747,Z 140.857,A -85,B 0,C 180,E1 -5892.192,E2 -5892.192} C_VEL
LIN {X 0,Y 502.78,Z 140.856,A -85,B 0,C 180,E1 -5895.471,E2 -5895.471} C_VEL
LIN {X 0,Y 502.752,Z 140.864,A -85,B 0,C 180,E1 -5898.927,E2 -5898.927} C_VEL
LIN {X 0,Y 502.749,Z 140.857,A -85,B 0,C 180,E1 -5902.042,E2 -5902.042} C_VEL
LIN {X 0,Y 502.769,Z 140.859,A -85,B 0,C 180,E1 -5905.032,E2 -5905.032} C_VEL
LIN {X 0,Y 502.758,Z 140.854,A -85,B 0,C 180,E1 -5907.913,E2 -5907.913} C_VEL
LIN {X 0,Y 502.755,Z 140.859,A -85,B 0,C 180,E1 -5910.708,E2 -5910.708} C_VEL
LIN {X 0,Y 502.773,Z 140.853,A -85,B 0,C 180,E1 -5913.461,E2 -5913.461} C_VEL
LIN {X 0,Y 502.749,Z 140.855,A -85,B 0,C 180,E1 -5916.084,E2 -5916.084} C_VEL
LIN {X 0,Y 502.759,Z 140.857,A -85,B 0,C 180,E1 -5918.688,E2 -5918.688} C_VEL
LIN {X 0,Y 502.791,Z 140.852,A -85,B 0,C 180,E1 -5921.899,E2 -5921.899} C_VEL
LIN {X 0,Y 502.796,Z 140.854,A -85,B 0,C 180,E1 -5924.683,E2 -5924.683} C_VEL
LIN {X 0,Y 502.844,Z 140.848,A -85,B 0,C 180,E1 -5928.06,E2 -5928.06} C_VEL
LIN {X 0,Y 502.839,Z 140.844,A -85,B 0,C 180,E1 -5931.156,E2 -5931.156} C_VEL
LIN {X 0,Y 502.853,Z 140.839,A -85,B 0,C 180,E1 -5933.58,E2 -5933.58} C_VEL
LIN {X 0,Y 502.746,Z 140.861,A -85,B 0,C 180,E1 -5935.992,E2 -5935.992} C_VEL
LIN {X 0,Y 503.011,Z 140.822,A -85,B 0,C 180,E1 -5937.598,E2 -5937.598} C_VEL
LIN {X 0,Y 503.007,Z 140.829,A -85,B 0,C 180,E1 -5940,E2 -5940} C_VEL
LIN {X 0,Y 503.012,Z 140.827,A -85,B 0,C 180,E1 -5942.402,E2 -5942.402} C_VEL
LIN {X 0,Y 502.895,Z 140.84,A -85,B 0,C 180,E1 -5945.614,E2 -5945.614} C_VEL
LIN {X 0,Y 502.851,Z 140.85,A -85,B 0,C 180,E1 -5948.034,E2 -5948.034} C_VEL
LIN {X 0,Y 502.841,Z 140.846,A -85,B 0,C 180,E1 -5951.284,E2 -5951.284} C_VEL
LIN {X 0,Y 502.829,Z 140.847,A -85,B 0,C 180,E1 -5954.571,E2 -5954.571} C_VEL
LIN {X 0,Y 502.788,Z 140.857,A -85,B 0,C 180,E1 -5957.91,E2 -5957.91} C_VEL
LIN {X 0,Y 502.806,Z 140.849,A -85,B 0,C 180,E1 -5960.527,E2 -5960.527} C_VEL
LIN {X 0,Y 502.786,Z 140.853,A -85,B 0,C 180,E1 -5963.041,E2 -5963.041} C_VEL
LIN {X 0,Y 502.781,Z 140.861,A -85,B 0,C 180,E1 -5965.679,E2 -5965.679} C_VEL
LIN {X 0,Y 502.772,Z 140.856,A -85,B 0,C 180,E1 -5968.377,E2 -5968.377} C_VEL
LIN {X 0,Y 502.789,Z 140.859,A -85,B 0,C 180,E1 -5971.497,E2 -5971.497} C_VEL
LIN {X 0,Y 502.791,Z 140.854,A -85,B 0,C 180,E1 -5974.441,E2 -5974.441} C_VEL
LIN {X 0,Y 502.812,Z 140.889,A -85,B 0,C 180,E1 -5977.182,E2 -5977.182} C_VEL
LIN {X 0,Y 503.692,Z 146.269,A -85,B 0,C 180,E1 -5978.245,E2 -5978.245} C_VEL
LIN {X 0,Y 503.46,Z 160.968,A -85,B 0,C 180,E1 -5981.003,E2 -5981.003} C_VEL
LIN {X 0,Y 503.347,Z 167.63,A -85,B 0,C 180,E1 -5982.25,E2 -5982.25} C_VEL
LIN {X 0,Y 505.506,Z 179.614,A -85,B 0,C 180,E1 -5982.502,E2 -5982.502} C_VEL
LIN {X 0,Y 504.841,Z 275.401,A -85,B 0,C 180,E1 -5983.907,E2 -5983.907} C_VEL
LIN {X 0,Y 504.654,Z 287.254,A -85,B 0,C 180,E1 -5984.223,E2 -5984.223} C_VEL
LIN {X 0,Y 503.88,Z 292.997,A -85,B 0,C 180,E1 -5984.407,E2 -5984.407} C_VEL
LIN {X 0,Y 500.897,Z 302.11,A -85,B 0,C 180,E1 -5984.728,E2 -5984.728} C_VEL
LIN {X 0,Y 497.855,Z 310.807,A -85,B 0,C 180,E1 -5985.123,E2 -5985.123} C_VEL
LIN {X 0,Y 497.007,Z 315.888,A -85,B 0,C 180,E1 -5985.428,E2 -5985.428} C_VEL
LIN {X 0,Y 496.637,Z 326.881,A -85,B 0,C 180,E1 -5986.26,E2 -5986.26} C_VEL
LIN {X 0,Y 496.306,Z 336.624,A -85,B 0,C 180,E1 -5987.179,E2 -5987.179} C_VEL
LIN {X 0,Y 495.939,Z 345.806,A -85,B 0,C 180,E1 -5988.237,E2 -5988.237} C_VEL
LIN {X 0,Y 495.635,Z 354.52,A -85,B 0,C 180,E1 -5989.479,E2 -5989.479} C_VEL
LIN {X 0,Y 495.37,Z 362.074,A -85,B 0,C 180,E1 -5990.848,E2 -5990.848} C_VEL
LIN {X 0,Y 495.237,Z 366.662,A -85,B 0,C 180,E1 -5991.879,E2 -5991.879} C_VEL
LIN {X 0,Y 495.098,Z 371.918,A -85,B 0,C 180,E1 -5993.402,E2 -5993.402} C_VEL
LIN {X 0,Y 494.998,Z 374.464,A -85,B 0,C 180,E1 -5994.4,E2 -5994.4} C_VEL
LIN {X 0,Y 494.929,Z 376.469,A -85,B 0,C 180,E1 -5995.447,E2 -5995.447} C_VEL
LIN {X 0,Y 494.884,Z 378.084,A -85,B 0,C 180,E1 -5996.917,E2 -5996.917} C_VEL
LIN {X 0,Y 494.898,Z 378.405,A -85,B 0,C 180,E1 -5998.436,E2 -5998.436} C_VEL
LIN {X 0,Y 494.943,Z 377.303,A -85,B 0,C 180,E1 -6000.018,E2 -6000.018} C_VEL
LIN {X 0,Y 495.014,Z 374.463,A -85,B 0,C 180,E1 -6001.673,E2 -6001.673} C_VEL
LIN {X 0,Y 495.102,Z 370.979,A -85,B 0,C 180,E1 -6002.984,E2 -6002.984} C_VEL
LIN {X 0,Y 495.272,Z 366.037,A -85,B 0,C 180,E1 -6004.354,E2 -6004.354} C_VEL
LIN {X 0,Y 495.424,Z 359.637,A -85,B 0,C 180,E1 -6005.708,E2 -6005.708} C_VEL
LIN {X 0,Y 495.64,Z 352.452,A -85,B 0,C 180,E1 -6006.916,E2 -6006.916} C_VEL
LIN {X 0,Y 496.007,Z 343.23,A -85,B 0,C 180,E1 -6008.164,E2 -6008.164} C_VEL
LIN {X 0,Y 496.393,Z 332.927,A -85,B 0,C 180,E1 -6009.27,E2 -6009.27} C_VEL
LIN {X 0,Y 496.729,Z 322.809,A -85,B 0,C 180,E1 -6010.149,E2 -6010.149} C_VEL
LIN {X 0,Y 497.2,Z 311.716,A -85,B 0,C 180,E1 -6010.921,E2 -6010.921} C_VEL
LIN {X 0,Y 497.436,Z 300.13,A -85,B 0,C 180,E1 -6011.549,E2 -6011.549} C_VEL
LIN {X 0,Y 497.762,Z 287.189,A -85,B 0,C 180,E1 -6012.063,E2 -6012.063} C_VEL
LIN {X 0,Y 497.978,Z 274.991,A -85,B 0,C 180,E1 -6012.389,E2 -6012.389} C_VEL
LIN {X 0,Y 498.525,Z 179.307,A -85,B 0,C 180,E1 -6013.811,E2 -6013.811} C_VEL
LIN {X 0,Y 496.315,Z 167.677,A -85,B 0,C 180,E1 -6014.076,E2 -6014.076} C_VEL
LIN {X 0,Y 496.776,Z 151.76,A -85,B 0,C 180,E1 -6017.18,E2 -6017.18} C_VEL
LIN {X 0,Y 496.708,Z 146.821,A -85,B 0,C 180,E1 -6018.161,E2 -6018.161} C_VEL
LIN {X 0,Y 495.821,Z 141.726,A -85,B 0,C 180,E1 -6019.226,E2 -6019.226} C_VEL
LIN {X 0,Y 495.833,Z 141.721,A -85,B 0,C 180,E1 -6021.851,E2 -6021.851} C_VEL
LIN {X 0,Y 495.832,Z 141.718,A -85,B 0,C 180,E1 -6025.121,E2 -6025.121} C_VEL
LIN {X 0,Y 495.988,Z 141.698,A -85,B 0,C 180,E1 -6027.564,E2 -6027.564} C_VEL
LIN {X 0,Y 495.943,Z 141.706,A -85,B 0,C 180,E1 -6030.812,E2 -6030.812} C_VEL
LIN {X 0,Y 495.981,Z 141.706,A -85,B 0,C 180,E1 -6032.436,E2 -6032.436} C_VEL
LIN {X 0,Y 495.858,Z 141.716,A -85,B 0,C 180,E1 -6035.694,E2 -6035.694} C_VEL
LIN {X 0,Y 495.818,Z 141.727,A -85,B 0,C 180,E1 -6038.149,E2 -6038.149} C_VEL
LIN {X 0,Y 495.854,Z 141.715,A -85,B 0,C 180,E1 -6041.445,E2 -6041.445} C_VEL
LIN {X 0,Y 495.782,Z 141.724,A -85,B 0,C 180,E1 -6044.783,E2 -6044.783} C_VEL
LIN {X 0,Y 495.775,Z 141.729,A -85,B 0,C 180,E1 -6048.235,E2 -6048.235} C_VEL
LIN {X 0,Y 495.777,Z 141.724,A -85,B 0,C 180,E1 -6050.756,E2 -6050.756} C_VEL
LIN {X 0,Y 495.741,Z 141.731,A -85,B 0,C 180,E1 -6053.388,E2 -6053.388} C_VEL
LIN {X 0,Y 495.742,Z 141.728,A -85,B 0,C 180,E1 -6056.73,E2 -6056.73} C_VEL
LIN {X 0,Y 495.76,Z 141.734,A -85,B 0,C 180,E1 -6059.747,E2 -6059.747} C_VEL
LIN {X 0,Y 495.755,Z 141.727,A -85,B 0,C 180,E1 -6062.596,E2 -6062.596} C_VEL
LIN {X 0,Y 495.746,Z 141.736,A -85,B 0,C 180,E1 -6065.538,E2 -6065.538} C_VEL
LIN {X 0,Y 495.762,Z 141.727,A -85,B 0,C 180,E1 -6068.768,E2 -6068.768} C_VEL
LIN {X 0,Y 495.726,Z 141.733,A -85,B 0,C 180,E1 -6071.785,E2 -6071.785} C_VEL
LIN {X 0,Y 495.74,Z 141.735,A -85,B 0,C 180,E1 -6075.141,E2 -6075.141} C_VEL
LIN {X 0,Y 495.726,Z 141.73,A -85,B 0,C 180,E1 -6078.216,E2 -6078.216} C_VEL
LIN {X 0,Y 495.749,Z 141.732,A -85,B 0,C 180,E1 -6081.408,E2 -6081.408} C_VEL
LIN {X 0,Y 495.746,Z 141.729,A -85,B 0,C 180,E1 -6084.462,E2 -6084.462} C_VEL
LIN {X 0,Y 495.754,Z 141.73,A -85,B 0,C 180,E1 -6087.404,E2 -6087.404} C_VEL
LIN {X 0,Y 495.743,Z 141.729,A -85,B 0,C 180,E1 -6090.252,E2 -6090.252} C_VEL
LIN {X 0,Y 495.743,Z 141.731,A -85,B 0,C 180,E1 -6093.271,E2 -6093.271} C_VEL
LIN {X 0,Y 495.738,Z 141.735,A -85,B 0,C 180,E1 -6096.612,E2 -6096.612} C_VEL
LIN {X 0,Y 495.783,Z 141.724,A -85,B 0,C 180,E1 -6099.324,E2 -6099.324} C_VEL
LIN {X 0,Y 495.765,Z 141.726,A -85,B 0,C 180,E1 -6101.828,E2 -6101.828} C_VEL
LIN {X 0,Y 495.778,Z 141.725,A -85,B 0,C 180,E1 -6105.217,E2 -6105.217} C_VEL
LIN {X 0,Y 495.855,Z 141.722,A -85,B 0,C 180,E1 -6108.555,E2 -6108.555} C_VEL
LIN {X 0,Y 495.815,Z 141.721,A -85,B 0,C 180,E1 -6111.851,E2 -6111.851} C_VEL
LIN {X 0,Y 495.855,Z 141.723,A -85,B 0,C 180,E1 -6114.306,E2 -6114.306} C_VEL
LIN {X 0,Y 495.979,Z 141.7,A -85,B 0,C 180,E1 -6117.564,E2 -6117.564} C_VEL
LIN {X 0,Y 495.976,Z 141.705,A -85,B 0,C 180,E1 -6120,E2 -6120} C_VEL
LIN {X 0,Y 495.979,Z 141.703,A -85,B 0,C 180,E1 -6122.436,E2 -6122.436} C_VEL
LIN {X 0,Y 495.853,Z 141.718,A -85,B 0,C 180,E1 -6125.694,E2 -6125.694} C_VEL
LIN {X 0,Y 495.814,Z 141.726,A -85,B 0,C 180,E1 -6128.149,E2 -6128.149} C_VEL
LIN {X 0,Y 495.825,Z 141.721,A -85,B 0,C 180,E1 -6131.446,E2 -6131.446} C_VEL
LIN {X 0,Y 495.757,Z 141.726,A -85,B 0,C 180,E1 -6134.784,E2 -6134.784} C_VEL
LIN {X 0,Y 495.751,Z 141.73,A -85,B 0,C 180,E1 -6138.226,E2 -6138.226} C_VEL
LIN {X 0,Y 495.726,Z 141.739,A -85,B 0,C 180,E1 -6141.63,E2 -6141.63} C_VEL
LIN {X 0,Y 495.704,Z 141.734,A -85,B 0,C 180,E1 -6144.278,E2 -6144.278} C_VEL
LIN {X 0,Y 495.721,Z 141.733,A -85,B 0,C 180,E1 -6146.98,E2 -6146.98} C_VEL
LIN {X 0,Y 495.698,Z 141.738,A -85,B 0,C 180,E1 -6149.751,E2 -6149.751} C_VEL
LIN {X 0,Y 495.727,Z 141.731,A -85,B 0,C 180,E1 -6152.597,E2 -6152.597} C_VEL
LIN {X 0,Y 495.729,Z 141.735,A -85,B 0,C 180,E1 -6155.539,E2 -6155.539} C_VEL
LIN {X 0,Y 495.735,Z 141.732,A -85,B 0,C 180,E1 -6158.763,E2 -6158.763} C_VEL
LIN {X 0,Y 495.725,Z 141.732,A -85,B 0,C 180,E1 -6161.785,E2 -6161.785} C_VEL
LIN {X 0,Y 495.733,Z 141.738,A -85,B 0,C 180,E1 -6165.142,E2 -6165.142} C_VEL
LIN {X 0,Y 495.724,Z 141.731,A -85,B 0,C 180,E1 -6168.215,E2 -6168.215} C_VEL
LIN {X 0,Y 495.718,Z 141.734,A -85,B 0,C 180,E1 -6171.405,E2 -6171.405} C_VEL
LIN {X 0,Y 495.72,Z 141.734,A -85,B 0,C 180,E1 -6174.46,E2 -6174.46} C_VEL
LIN {X 0,Y 495.726,Z 141.732,A -85,B 0,C 180,E1 -6177.402,E2 -6177.402} C_VEL
LIN {X 0,Y 495.697,Z 141.739,A -85,B 0,C 180,E1 -6180.249,E2 -6180.249} C_VEL
LIN {X 0,Y 495.722,Z 141.736,A -85,B 0,C 180,E1 -6183.275,E2 -6183.275} C_VEL
LIN {X 0,Y 495.746,Z 141.821,A -85,B 0,C 180,E1 -6185.175,E2 -6185.175} C_VEL
LIN {X 0,Y 497.463,Z 150.915,A -85,B 0,C 180,E1 -6186.842,E2 -6186.842} C_VEL
LIN {X 0,Y 497.182,Z 163.66,A -85,B 0,C 180,E1 -6189.024,E2 -6189.024} C_VEL
LIN {X 0,Y 496.607,Z 180.518,A -85,B 0,C 180,E1 -6191.86,E2 -6191.86} C_VEL
LIN {X 0,Y 496.251,Z 193.149,A -85,B 0,C 180,E1 -6193.963,E2 -6193.963} C_VEL
LIN {X 0,Y 498.471,Z 208.181,A -85,B 0,C 180,E1 -6194.267,E2 -6194.267} C_VEL
LIN {X 0,Y 497.929,Z 301.335,A -85,B 0,C 180,E1 -6195.647,E2 -6195.647} C_VEL
LIN {X 0,Y 497.661,Z 314.573,A -85,B 0,C 180,E1 -6196.005,E2 -6196.005} C_VEL
LIN {X 0,Y 497.28,Z 327.294,A -85,B 0,C 180,E1 -6196.515,E2 -6196.515} C_VEL
LIN {X 0,Y 496.94,Z 338.732,A -85,B 0,C 180,E1 -6197.138,E2 -6197.138} C_VEL
LIN {X 0,Y 496.54,Z 350.287,A -85,B 0,C 180,E1 -6197.95,E2 -6197.95} C_VEL
LIN {X 0,Y 496.226,Z 360.795,A -85,B 0,C 180,E1 -6198.874,E2 -6198.874} C_VEL
LIN {X 0,Y 495.824,Z 369.381,A -85,B 0,C 180,E1 -6199.794,E2 -6199.794} C_VEL
LIN {X 0,Y 495.585,Z 377.304,A -85,B 0,C 180,E1 -6200.82,E2 -6200.82} C_VEL
LIN {X 0,Y 495.33,Z 385.04,A -85,B 0,C 180,E1 -6202.048,E2 -6202.048} C_VEL
LIN {X 0,Y 495.172,Z 390.334,A -85,B 0,C 180,E1 -6203.071,E2 -6203.071} C_VEL
LIN {X 0,Y 495.117,Z 395.466,A -85,B 0,C 180,E1 -6204.298,E2 -6204.298} C_VEL
LIN {X 0,Y 495.006,Z 399.446,A -85,B 0,C 180,E1 -6205.521,E2 -6205.521} C_VEL
LIN {X 0,Y 495.041,Z 402.386,A -85,B 0,C 180,E1 -6206.745,E2 -6206.745} C_VEL
LIN {X 0,Y 494.998,Z 403.785,A -85,B 0,C 180,E1 -6207.559,E2 -6207.559} C_VEL
LIN {X 0,Y 494.962,Z 404.78,A -85,B 0,C 180,E1 -6208.373,E2 -6208.373} C_VEL
LIN {X 0,Y 494.902,Z 405.6,A -85,B 0,C 180,E1 -6210,E2 -6210} C_VEL
LIN {X 0,Y 494.962,Z 404.769,A -85,B 0,C 180,E1 -6211.627,E2 -6211.627} C_VEL
LIN {X 0,Y 494.998,Z 403.768,A -85,B 0,C 180,E1 -6212.441,E2 -6212.441} C_VEL
LIN {X 0,Y 495.041,Z 402.364,A -85,B 0,C 180,E1 -6213.255,E2 -6213.255} C_VEL
LIN {X 0,Y 495.006,Z 399.41,A -85,B 0,C 180,E1 -6214.479,E2 -6214.479} C_VEL
LIN {X 0,Y 495.115,Z 395.418,A -85,B 0,C 180,E1 -6215.703,E2 -6215.703} C_VEL
LIN {X 0,Y 495.253,Z 389.274,A -85,B 0,C 180,E1 -6217.133,E2 -6217.133} C_VEL
LIN {X 0,Y 495.418,Z 382.562,A -85,B 0,C 180,E1 -6218.361,E2 -6218.361} C_VEL
LIN {X 0,Y 495.686,Z 374.236,A -85,B 0,C 180,E1 -6219.59,E2 -6219.59} C_VEL
LIN {X 0,Y 495.968,Z 365.689,A -85,B 0,C 180,E1 -6220.615,E2 -6220.615} C_VEL
LIN {X 0,Y 496.378,Z 355.133,A -85,B 0,C 180,E1 -6221.64,E2 -6221.64} C_VEL
LIN {X 0,Y 496.749,Z 343.835,A -85,B 0,C 180,E1 -6222.522,E2 -6222.522} C_VEL
LIN {X 0,Y 497.081,Z 333.215,A -85,B 0,C 180,E1 -6223.179,E2 -6223.179} C_VEL
LIN {X 0,Y 497.42,Z 321.367,A -85,B 0,C 180,E1 -6223.742,E2 -6223.742} C_VEL
LIN {X 0,Y 497.795,Z 307.708,A -85,B 0,C 180,E1 -6224.2,E2 -6224.2} C_VEL
LIN {X 0,Y 498.047,Z 293.758,A -85,B 0,C 180,E1 -6224.48,E2 -6224.48} C_VEL
LIN {X 0,Y 498.44,Z 207.128,A -85,B 0,C 180,E1 -6225.752,E2 -6225.752} C_VEL
LIN {X 0,Y 496.24,Z 192.809,A -85,B 0,C 180,E1 -6226.055,E2 -6226.055} C_VEL
LIN {X 0,Y 496.779,Z 173.801,A -85,B 0,C 180,E1 -6229.203,E2 -6229.203} C_VEL
LIN {X 0,Y 497.262,Z 157.165,A -85,B 0,C 180,E1 -6231.996,E2 -6231.996} C_VEL
LIN {X 0,Y 497.383,Z 150.499,A -85,B 0,C 180,E1 -6233.13,E2 -6233.13} C_VEL
LIN {X 0,Y 495.73,Z 141.737,A -85,B 0,C 180,E1 -6234.733,E2 -6234.733} C_VEL
LIN {X 0,Y 495.71,Z 141.739,A -85,B 0,C 180,E1 -6237.896,E2 -6237.896} C_VEL
LIN {X 0,Y 495.71,Z 141.738,A -85,B 0,C 180,E1 -6240.69,E2 -6240.69} C_VEL
LIN {X 0,Y 495.724,Z 141.738,A -85,B 0,C 180,E1 -6243.567,E2 -6243.567} C_VEL
LIN {X 0,Y 495.677,Z 141.739,A -85,B 0,C 180,E1 -6246.549,E2 -6246.549} C_VEL
LIN {X 0,Y 495.708,Z 141.736,A -85,B 0,C 180,E1 -6249.643,E2 -6249.643} C_VEL
LIN {X 0,Y 495.691,Z 141.742,A -85,B 0,C 180,E1 -6252.887,E2 -6252.887} C_VEL
LIN {X 0,Y 495.715,Z 141.734,A -85,B 0,C 180,E1 -6255.997,E2 -6255.997} C_VEL
LIN {X 0,Y 495.71,Z 141.735,A -85,B 0,C 180,E1 -6259.294,E2 -6259.294} C_VEL
LIN {X 0,Y 495.711,Z 141.735,A -85,B 0,C 180,E1 -6261.405,E2 -6261.405} C_VEL
LIN {X 0,Y 495.72,Z 141.734,A -85,B 0,C 180,E1 -6264.46,E2 -6264.46} C_VEL
LIN {X 0,Y 495.726,Z 141.731,A -85,B 0,C 180,E1 -6267.402,E2 -6267.402} C_VEL
LIN {X 0,Y 495.698,Z 141.736,A -85,B 0,C 180,E1 -6270.249,E2 -6270.249} C_VEL
LIN {X 0,Y 495.724,Z 141.732,A -85,B 0,C 180,E1 -6273.275,E2 -6273.275} C_VEL
LIN {X 0,Y 495.7,Z 141.731,A -85,B 0,C 180,E1 -6275.722,E2 -6275.722} C_VEL
LIN {X 0,Y 495.726,Z 141.736,A -85,B 0,C 180,E1 -6278.37,E2 -6278.37} C_VEL
LIN {X 0,Y 495.739,Z 141.73,A -85,B 0,C 180,E1 -6281.827,E2 -6281.827} C_VEL
LIN {X 0,Y 495.747,Z 141.727,A -85,B 0,C 180,E1 -6285.216,E2 -6285.216} C_VEL
LIN {X 0,Y 495.818,Z 141.721,A -85,B 0,C 180,E1 -6288.554,E2 -6288.554} C_VEL
LIN {X 0,Y 495.814,Z 141.722,A -85,B 0,C 180,E1 -6291.851,E2 -6291.851} C_VEL
LIN {X 0,Y 495.847,Z 141.72,A -85,B 0,C 180,E1 -6294.306,E2 -6294.306} C_VEL
LIN {X 0,Y 495.978,Z 141.698,A -85,B 0,C 180,E1 -6297.564,E2 -6297.564} C_VEL
LIN {X 0,Y 495.976,Z 141.705,A -85,B 0,C 180,E1 -6300,E2 -6300} C_VEL
LIN {X 0,Y 495.979,Z 141.703,A -85,B 0,C 180,E1 -6302.436,E2 -6302.436} C_VEL
LIN {X 0,Y 495.854,Z 141.718,A -85,B 0,C 180,E1 -6305.694,E2 -6305.694} C_VEL
LIN {X 0,Y 495.815,Z 141.725,A -85,B 0,C 180,E1 -6308.149,E2 -6308.149} C_VEL
LIN {X 0,Y 495.826,Z 141.721,A -85,B 0,C 180,E1 -6311.446,E2 -6311.446} C_VEL
LIN {X 0,Y 495.78,Z 141.725,A -85,B 0,C 180,E1 -6314.783,E2 -6314.783} C_VEL
LIN {X 0,Y 495.752,Z 141.731,A -85,B 0,C 180,E1 -6318.226,E2 -6318.226} C_VEL
LIN {X 0,Y 495.75,Z 141.728,A -85,B 0,C 180,E1 -6320.758,E2 -6320.758} C_VEL
LIN {X 0,Y 495.739,Z 141.734,A -85,B 0,C 180,E1 -6323.388,E2 -6323.388} C_VEL
LIN {X 0,Y 495.721,Z 141.737,A -85,B 0,C 180,E1 -6326.072,E2 -6326.072} C_VEL
LIN {X 0,Y 495.72,Z 141.734,A -85,B 0,C 180,E1 -6328.818,E2 -6328.818} C_VEL
LIN {X 0,Y 495.753,Z 141.735,A -85,B 0,C 180,E1 -6331.724,E2 -6331.724} C_VEL
LIN {X 0,Y 495.763,Z 141.73,A -85,B 0,C 180,E1 -6334.692,E2 -6334.692} C_VEL
LIN {X 0,Y 495.821,Z 141.857,A -85,B 0,C 180,E1 -6337.043,E2 -6337.043} C_VEL
LIN {X 0,Y 496.749,Z 147.897,A -85,B 0,C 180,E1 -6338.241,E2 -6338.241} C_VEL
LIN {X 0,Y 496.446,Z 163.421,A -85,B 0,C 180,E1 -6341.191,E2 -6341.191} C_VEL
LIN {X 0,Y 496.366,Z 167.889,A -85,B 0,C 180,E1 -6342.025,E2 -6342.025} C_VEL
LIN {X 0,Y 498.659,Z 180.868,A -85,B 0,C 180,E1 -6342.298,E2 -6342.298} C_VEL
LIN {X 0,Y 498.004,Z 275.055,A -85,B 0,C 180,E1 -6343.697,E2 -6343.697} C_VEL
LIN {X 0,Y 497.765,Z 288.005,A -85,B 0,C 180,E1 -6344.048,E2 -6344.048} C_VEL
LIN {X 0,Y 497.493,Z 300.671,A -85,B 0,C 180,E1 -6344.559,E2 -6344.559} C_VEL
LIN {X 0,Y 497.083,Z 312.835,A -85,B 0,C 180,E1 -6345.229,E2 -6345.229} C_VEL
LIN {X 0,Y 497.007,Z 315.888,A -85,B 0,C 180,E1 -6345.428,E2 -6345.428} C_VEL
LIN {X 0,Y 496.177,Z 320.973,A -85,B 0,C 180,E1 -6345.762,E2 -6345.762} C_VEL
LIN {X 0,Y 493.13,Z 328.981,A -85,B 0,C 180,E1 -6346.339,E2 -6346.339} C_VEL
LIN {X 0,Y 490.034,Z 336.497,A -85,B 0,C 180,E1 -6346.999,E2 -6346.999} C_VEL
LIN {X 0,Y 489.134,Z 340.808,A -85,B 0,C 180,E1 -6347.46,E2 -6347.46} C_VEL
LIN {X 0,Y 488.757,Z 349.646,A -85,B 0,C 180,E1 -6348.589,E2 -6348.589} C_VEL
LIN {X 0,Y 488.48,Z 358.113,A -85,B 0,C 180,E1 -6349.937,E2 -6349.937} C_VEL
LIN {X 0,Y 488.269,Z 363.557,A -85,B 0,C 180,E1 -6351.011,E2 -6351.011} C_VEL
LIN {X 0,Y 488.105,Z 369.02,A -85,B 0,C 180,E1 -6352.366,E2 -6352.366} C_VEL
LIN {X 0,Y 487.944,Z 373.374,A -85,B 0,C 180,E1 -6353.805,E2 -6353.805} C_VEL
LIN {X 0,Y 487.838,Z 376.313,A -85,B 0,C 180,E1 -6355.202,E2 -6355.202} C_VEL
LIN {X 0,Y 487.785,Z 378.225,A -85,B 0,C 180,E1 -6356.804,E2 -6356.804} C_VEL
LIN {X 0,Y 487.794,Z 378.644,A -85,B 0,C 180,E1 -6358.218,E2 -6358.218} C_VEL
LIN {X 0,Y 487.862,Z 377.734,A -85,B 0,C 180,E1 -6359.808,E2 -6359.808} C_VEL
LIN {X 0,Y 487.865,Z 376.643,A -85,B 0,C 180,E1 -6360.673,E2 -6360.673} C_VEL
LIN {X 0,Y 487.94,Z 373.831,A -85,B 0,C 180,E1 -6362.088,E2 -6362.088} C_VEL
LIN {X 0,Y 488.066,Z 369.77,A -85,B 0,C 180,E1 -6363.487,E2 -6363.487} C_VEL
LIN {X 0,Y 488.262,Z 364.785,A -85,B 0,C 180,E1 -6364.779,E2 -6364.779} C_VEL
LIN {X 0,Y 488.444,Z 358.748,A -85,B 0,C 180,E1 -6366.016,E2 -6366.016} C_VEL
LIN {X 0,Y 488.639,Z 351.94,A -85,B 0,C 180,E1 -6367.149,E2 -6367.149} C_VEL
LIN {X 0,Y 489.008,Z 343.638,A -85,B 0,C 180,E1 -6368.279,E2 -6368.279} C_VEL
LIN {X 0,Y 489.42,Z 333.386,A -85,B 0,C 180,E1 -6369.401,E2 -6369.401} C_VEL
LIN {X 0,Y 489.767,Z 323.326,A -85,B 0,C 180,E1 -6370.292,E2 -6370.292} C_VEL
LIN {X 0,Y 490.274,Z 311.859,A -85,B 0,C 180,E1 -6371.103,E2 -6371.103} C_VEL
LIN {X 0,Y 490.544,Z 300.343,A -85,B 0,C 180,E1 -6371.735,E2 -6371.735} C_VEL
LIN {X 0,Y 490.882,Z 287.29,A -85,B 0,C 180,E1 -6372.261,E2 -6372.261} C_VEL
LIN {X 0,Y 491.113,Z 274.689,A -85,B 0,C 180,E1 -6372.6,E2 -6372.6} C_VEL
LIN {X 0,Y 491.764,Z 181.151,A -85,B 0,C 180,E1 -6374.005,E2 -6374.005} C_VEL
LIN {X 0,Y 489.351,Z 167.877,A -85,B 0,C 180,E1 -6374.301,E2 -6374.301} C_VEL
LIN {X 0,Y 489.864,Z 151.302,A -85,B 0,C 180,E1 -6377.572,E2 -6377.572} C_VEL
LIN {X 0,Y 489.585,Z 147.196,A -85,B 0,C 180,E1 -6378.406,E2 -6378.406} C_VEL
LIN {X 0,Y 488.767,Z 142.604,A -85,B 0,C 180,E1 -6379.384,E2 -6379.384} C_VEL
LIN {X 0,Y 488.805,Z 142.599,A -85,B 0,C 180,E1 -6382.565,E2 -6382.565} C_VEL
LIN {X 0,Y 488.801,Z 142.595,A -85,B 0,C 180,E1 -6385.051,E2 -6385.051} C_VEL
LIN {X 0,Y 488.955,Z 142.574,A -85,B 0,C 180,E1 -6387.529,E2 -6387.529} C_VEL
LIN {X 0,Y 488.896,Z 142.584,A -85,B 0,C 180,E1 -6390.824,E2 -6390.824} C_VEL
LIN {X 0,Y 488.947,Z 142.581,A -85,B 0,C 180,E1 -6392.471,E2 -6392.471} C_VEL
LIN {X 0,Y 488.818,Z 142.593,A -85,B 0,C 180,E1 -6395.776,E2 -6395.776} C_VEL
LIN {X 0,Y 488.766,Z 142.605,A -85,B 0,C 180,E1 -6398.267,E2 -6398.267} C_VEL
LIN {X 0,Y 488.808,Z 142.594,A -85,B 0,C 180,E1 -6401.612,E2 -6401.612} C_VEL
LIN {X 0,Y 488.752,Z 142.599,A -85,B 0,C 180,E1 -6405.001,E2 -6405.001} C_VEL
LIN {X 0,Y 488.747,Z 142.602,A -85,B 0,C 180,E1 -6408.443,E2 -6408.443} C_VEL
LIN {X 0,Y 488.709,Z 142.605,A -85,B 0,C 180,E1 -6411.071,E2 -6411.071} C_VEL
LIN {X 0,Y 488.673,Z 142.617,A -85,B 0,C 180,E1 -6413.747,E2 -6413.747} C_VEL
LIN {X 0,Y 488.701,Z 142.606,A -85,B 0,C 180,E1 -6416.922,E2 -6416.922} C_VEL
LIN {X 0,Y 488.721,Z 142.605,A -85,B 0,C 180,E1 -6420.22,E2 -6420.22} C_VEL
LIN {X 0,Y 488.713,Z 142.611,A -85,B 0,C 180,E1 -6423.48,E2 -6423.48} C_VEL
LIN {X 0,Y 488.675,Z 142.609,A -85,B 0,C 180,E1 -6426.353,E2 -6426.353} C_VEL
LIN {X 0,Y 488.697,Z 142.612,A -85,B 0,C 180,E1 -6429.255,E2 -6429.255} C_VEL
LIN {X 0,Y 488.653,Z 142.612,A -85,B 0,C 180,E1 -6432.53,E2 -6432.53} C_VEL
LIN {X 0,Y 488.704,Z 142.613,A -85,B 0,C 180,E1 -6435.197,E2 -6435.197} C_VEL
LIN {X 0,Y 488.665,Z 142.611,A -85,B 0,C 180,E1 -6438.58,E2 -6438.58} C_VEL
LIN {X 0,Y 488.701,Z 142.611,A -85,B 0,C 180,E1 -6440.948,E2 -6440.948} C_VEL
LIN {X 0,Y 488.672,Z 142.609,A -85,B 0,C 180,E1 -6443.867,E2 -6443.867} C_VEL
LIN {X 0,Y 488.705,Z 142.612,A -85,B 0,C 180,E1 -6446.874,E2 -6446.874} C_VEL
LIN {X 0,Y 488.707,Z 142.605,A -85,B 0,C 180,E1 -6449.779,E2 -6449.779} C_VEL
LIN {X 0,Y 488.702,Z 142.611,A -85,B 0,C 180,E1 -6453.078,E2 -6453.078} C_VEL
LIN {X 0,Y 488.699,Z 142.607,A -85,B 0,C 180,E1 -6455.351,E2 -6455.351} C_VEL
LIN {X 0,Y 488.691,Z 142.608,A -85,B 0,C 180,E1 -6458.043,E2 -6458.043} C_VEL
LIN {X 0,Y 488.731,Z 142.61,A -85,B 0,C 180,E1 -6460.686,E2 -6460.686} C_VEL
LIN {X 0,Y 488.674,Z 142.61,A -85,B 0,C 180,E1 -6463.283,E2 -6463.283} C_VEL
LIN {X 0,Y 488.716,Z 142.604,A -85,B 0,C 180,E1 -6465.849,E2 -6465.849} C_VEL
LIN {X 0,Y 488.81,Z 142.599,A -85,B 0,C 180,E1 -6468.388,E2 -6468.388} C_VEL
LIN {X 0,Y 488.762,Z 142.599,A -85,B 0,C 180,E1 -6471.733,E2 -6471.733} C_VEL
LIN {X 0,Y 488.815,Z 142.598,A -85,B 0,C 180,E1 -6474.224,E2 -6474.224} C_VEL
LIN {X 0,Y 488.945,Z 142.576,A -85,B 0,C 180,E1 -6477.529,E2 -6477.529} C_VEL
LIN {X 0,Y 488.945,Z 142.581,A -85,B 0,C 180,E1 -6480,E2 -6480} C_VEL
LIN {X 0,Y 488.945,Z 142.579,A -85,B 0,C 180,E1 -6482.471,E2 -6482.471} C_VEL
LIN {X 0,Y 488.814,Z 142.596,A -85,B 0,C 180,E1 -6485.776,E2 -6485.776} C_VEL
LIN {X 0,Y 488.761,Z 142.603,A -85,B 0,C 180,E1 -6488.267,E2 -6488.267} C_VEL
LIN {X 0,Y 488.788,Z 142.599,A -85,B 0,C 180,E1 -6491.613,E2 -6491.613} C_VEL
LIN {X 0,Y 488.722,Z 142.603,A -85,B 0,C 180,E1 -6495.002,E2 -6495.002} C_VEL
LIN {X 0,Y 488.705,Z 142.606,A -85,B 0,C 180,E1 -6498.444,E2 -6498.444} C_VEL
LIN {X 0,Y 488.681,Z 142.609,A -85,B 0,C 180,E1 -6501.072,E2 -6501.072} C_VEL
LIN {X 0,Y 488.663,Z 142.617,A -85,B 0,C 180,E1 -6503.747,E2 -6503.747} C_VEL
LIN {X 0,Y 488.671,Z 142.609,A -85,B 0,C 180,E1 -6506.477,E2 -6506.477} C_VEL
LIN {X 0,Y 488.662,Z 142.616,A -85,B 0,C 180,E1 -6509.274,E2 -6509.274} C_VEL
LIN {X 0,Y 488.681,Z 142.609,A -85,B 0,C 180,E1 -6512.149,E2 -6512.149} C_VEL
LIN {X 0,Y 488.706,Z 142.61,A -85,B 0,C 180,E1 -6515.116,E2 -6515.116} C_VEL
LIN {X 0,Y 488.653,Z 142.612,A -85,B 0,C 180,E1 -6518.203,E2 -6518.203} C_VEL
LIN {X 0,Y 488.696,Z 142.606,A -85,B 0,C 180,E1 -6520.341,E2 -6520.341} C_VEL
LIN {X 0,Y 488.668,Z 142.612,A -85,B 0,C 180,E1 -6523.657,E2 -6523.657} C_VEL
LIN {X 0,Y 488.667,Z 142.61,A -85,B 0,C 180,E1 -6526.343,E2 -6526.343} C_VEL
LIN {X 0,Y 488.669,Z 142.61,A -85,B 0,C 180,E1 -6529.67,E2 -6529.67} C_VEL
LIN {X 0,Y 488.646,Z 142.614,A -85,B 0,C 180,E1 -6532.283,E2 -6532.283} C_VEL
LIN {X 0,Y 488.706,Z 142.61,A -85,B 0,C 180,E1 -6535.056,E2 -6535.056} C_VEL
LIN {X 0,Y 488.684,Z 142.608,A -85,B 0,C 180,E1 -6538.05,E2 -6538.05} C_VEL
LIN {X 0,Y 488.662,Z 142.614,A -85,B 0,C 180,E1 -6541.32,E2 -6541.32} C_VEL
LIN {X 0,Y 488.669,Z 142.614,A -85,B 0,C 180,E1 -6543.523,E2 -6543.523} C_VEL
LIN {X 0,Y 488.689,Z 142.717,A -85,B 0,C 180,E1 -6544.989,E2 -6544.989} C_VEL
LIN {X 0,Y 490.558,Z 153.01,A -85,B 0,C 180,E1 -6546.9,E2 -6546.9} C_VEL
LIN {X 0,Y 490.078,Z 167.648,A -85,B 0,C 180,E1 -6549.43,E2 -6549.43} C_VEL
LIN {X 0,Y 489.608,Z 181.583,A -85,B 0,C 180,E1 -6551.808,E2 -6551.808} C_VEL
LIN {X 0,Y 489.25,Z 192.981,A -85,B 0,C 180,E1 -6553.733,E2 -6553.733} C_VEL
LIN {X 0,Y 491.648,Z 209.249,A -85,B 0,C 180,E1 -6554.065,E2 -6554.065} C_VEL
LIN {X 0,Y 491.054,Z 300.935,A -85,B 0,C 180,E1 -6555.442,E2 -6555.442} C_VEL
LIN {X 0,Y 490.78,Z 314.246,A -85,B 0,C 180,E1 -6555.804,E2 -6555.804} C_VEL
LIN {X 0,Y 490.38,Z 327.004,A -85,B 0,C 180,E1 -6556.321,E2 -6556.321} C_VEL
LIN {X 0,Y 489.992,Z 338.351,A -85,B 0,C 180,E1 -6556.944,E2 -6556.944} C_VEL
LIN {X 0,Y 489.55,Z 350.044,A -85,B 0,C 180,E1 -6557.775,E2 -6557.775} C_VEL
LIN {X 0,Y 489.204,Z 360.565,A -85,B 0,C 180,E1 -6558.712,E2 -6558.712} C_VEL
LIN {X 0,Y 488.815,Z 369.161,A -85,B 0,C 180,E1 -6559.646,E2 -6559.646} C_VEL
LIN {X 0,Y 488.528,Z 377.089,A -85,B 0,C 180,E1 -6560.686,E2 -6560.686} C_VEL
LIN {X 0,Y 488.268,Z 384.832,A -85,B 0,C 180,E1 -6561.932,E2 -6561.932} C_VEL
LIN {X 0,Y 488.099,Z 390.129,A -85,B 0,C 180,E1 -6562.97,E2 -6562.97} C_VEL
LIN {X 0,Y 488.014,Z 395.265,A -85,B 0,C 180,E1 -6564.214,E2 -6564.214} C_VEL
LIN {X 0,Y 487.918,Z 399.248,A -85,B 0,C 180,E1 -6565.456,E2 -6565.456} C_VEL
LIN {X 0,Y 487.964,Z 402.19,A -85,B 0,C 180,E1 -6566.697,E2 -6566.697} C_VEL
LIN {X 0,Y 487.909,Z 403.589,A -85,B 0,C 180,E1 -6567.523,E2 -6567.523} C_VEL
LIN {X 0,Y 487.891,Z 404.586,A -85,B 0,C 180,E1 -6568.349,E2 -6568.349} C_VEL
LIN {X 0,Y 487.822,Z 405.406,A -85,B 0,C 180,E1 -6570,E2 -6570} C_VEL
LIN {X 0,Y 487.891,Z 404.574,A -85,B 0,C 180,E1 -6571.651,E2 -6571.651} C_VEL
LIN {X 0,Y 487.909,Z 403.572,A -85,B 0,C 180,E1 -6572.477,E2 -6572.477} C_VEL
LIN {X 0,Y 487.964,Z 402.167,A -85,B 0,C 180,E1 -6573.303,E2 -6573.303} C_VEL
LIN {X 0,Y 487.918,Z 399.211,A -85,B 0,C 180,E1 -6574.544,E2 -6574.544} C_VEL
LIN {X 0,Y 488.012,Z 395.215,A -85,B 0,C 180,E1 -6575.786,E2 -6575.786} C_VEL
LIN {X 0,Y 488.179,Z 389.068,A -85,B 0,C 180,E1 -6577.237,E2 -6577.237} C_VEL
LIN {X 0,Y 488.35,Z 382.353,A -85,B 0,C 180,E1 -6578.483,E2 -6578.483} C_VEL
LIN {X 0,Y 488.653,Z 374.026,A -85,B 0,C 180,E1 -6579.729,E2 -6579.729} C_VEL
LIN {X 0,Y 488.981,Z 365.479,A -85,B 0,C 180,E1 -6580.769,E2 -6580.769} C_VEL
LIN {X 0,Y 489.41,Z 354.923,A -85,B 0,C 180,E1 -6581.808,E2 -6581.808} C_VEL
LIN {X 0,Y 489.815,Z 343.184,A -85,B 0,C 180,E1 -6582.734,E2 -6582.734} C_VEL
LIN {X 0,Y 490.206,Z 331.034,A -85,B 0,C 180,E1 -6583.472,E2 -6583.472} C_VEL
LIN {X 0,Y 490.644,Z 318.55,A -85,B 0,C 180,E1 -6584.041,E2 -6584.041} C_VEL
LIN {X 0,Y 490.975,Z 305.582,A -85,B 0,C 180,E1 -6584.454,E2 -6584.454} C_VEL
LIN {X 0,Y 491.191,Z 289.994,A -85,B 0,C 180,E1 -6584.739,E2 -6584.739} C_VEL
LIN {X 0,Y 491.595,Z 207.936,A -85,B 0,C 180,E1 -6585.965,E2 -6585.965} C_VEL
LIN {X 0,Y 489.24,Z 192.574,A -85,B 0,C 180,E1 -6586.299,E2 -6586.299} C_VEL
LIN {X 0,Y 489.784,Z 174.886,A -85,B 0,C 180,E1 -6589.271,E2 -6589.271} C_VEL
LIN {X 0,Y 490.33,Z 158.252,A -85,B 0,C 180,E1 -6592.102,E2 -6592.102} C_VEL
LIN {X 0,Y 490.49,Z 152.507,A -85,B 0,C 180,E1 -6593.09,E2 -6593.09} C_VEL
LIN {X 0,Y 488.7,Z 142.614,A -85,B 0,C 180,E1 -6594.947,E2 -6594.947} C_VEL
LIN {X 0,Y 488.676,Z 142.617,A -85,B 0,C 180,E1 -6597.401,E2 -6597.401} C_VEL
LIN {X 0,Y 488.653,Z 142.617,A -85,B 0,C 180,E1 -6600.351,E2 -6600.351} C_VEL
LIN {X 0,Y 488.693,Z 142.615,A -85,B 0,C 180,E1 -6603.476,E2 -6603.476} C_VEL
LIN {X 0,Y 488.64,Z 142.614,A -85,B 0,C 180,E1 -6606.347,E2 -6606.347} C_VEL
LIN {X 0,Y 488.668,Z 142.617,A -85,B 0,C 180,E1 -6609.258,E2 -6609.258} C_VEL
LIN {X 0,Y 488.649,Z 142.615,A -85,B 0,C 180,E1 -6612.531,E2 -6612.531} C_VEL
LIN {X 0,Y 488.698,Z 142.614,A -85,B 0,C 180,E1 -6615.197,E2 -6615.197} C_VEL
LIN {X 0,Y 488.645,Z 142.617,A -85,B 0,C 180,E1 -6618.578,E2 -6618.578} C_VEL
LIN {X 0,Y 488.647,Z 142.613,A -85,B 0,C 180,E1 -6621.797,E2 -6621.797} C_VEL
LIN {X 0,Y 488.706,Z 142.61,A -85,B 0,C 180,E1 -6625.056,E2 -6625.056} C_VEL
LIN {X 0,Y 488.685,Z 142.607,A -85,B 0,C 180,E1 -6628.05,E2 -6628.05} C_VEL
LIN {X 0,Y 488.663,Z 142.61,A -85,B 0,C 180,E1 -6631.32,E2 -6631.32} C_VEL
LIN {X 0,Y 488.671,Z 142.609,A -85,B 0,C 180,E1 -6633.523,E2 -6633.523} C_VEL
LIN {X 0,Y 488.66,Z 142.612,A -85,B 0,C 180,E1 -6636.253,E2 -6636.253} C_VEL
LIN {X 0,Y 488.675,Z 142.605,A -85,B 0,C 180,E1 -6639.199,E2 -6639.199} C_VEL
LIN {X 0,Y 488.709,Z 142.605,A -85,B 0,C 180,E1 -6641.648,E2 -6641.648} C_VEL
LIN {X 0,Y 488.717,Z 142.604,A -85,B 0,C 180,E1 -6644.998,E2 -6644.998} C_VEL
LIN {X 0,Y 488.778,Z 142.599,A -85,B 0,C 180,E1 -6648.387,E2 -6648.387} C_VEL
LIN {X 0,Y 488.758,Z 142.6,A -85,B 0,C 180,E1 -6651.733,E2 -6651.733} C_VEL
LIN {X 0,Y 488.807,Z 142.595,A -85,B 0,C 180,E1 -6654.224,E2 -6654.224} C_VEL
LIN {X 0,Y 488.944,Z 142.574,A -85,B 0,C 180,E1 -6657.529,E2 -6657.529} C_VEL
LIN {X 0,Y 488.945,Z 142.581,A -85,B 0,C 180,E1 -6660,E2 -6660} C_VEL
LIN {X 0,Y 488.944,Z 142.579,A -85,B 0,C 180,E1 -6662.471,E2 -6662.471} C_VEL
LIN {X 0,Y 488.814,Z 142.596,A -85,B 0,C 180,E1 -6665.776,E2 -6665.776} C_VEL
LIN {X 0,Y 488.761,Z 142.602,A -85,B 0,C 180,E1 -6668.267,E2 -6668.267} C_VEL
LIN {X 0,Y 488.788,Z 142.6,A -85,B 0,C 180,E1 -6671.613,E2 -6671.613} C_VEL
LIN {X 0,Y 488.751,Z 142.6,A -85,B 0,C 180,E1 -6675.001,E2 -6675.001} C_VEL
LIN {X 0,Y 488.71,Z 142.606,A -85,B 0,C 180,E1 -6678.444,E2 -6678.444} C_VEL
LIN {X 0,Y 488.694,Z 142.608,A -85,B 0,C 180,E1 -6681.071,E2 -6681.071} C_VEL
LIN {X 0,Y 488.67,Z 142.618,A -85,B 0,C 180,E1 -6683.747,E2 -6683.747} C_VEL
LIN {X 0,Y 488.686,Z 142.611,A -85,B 0,C 180,E1 -6686.476,E2 -6686.476} C_VEL
LIN {X 0,Y 488.691,Z 142.614,A -85,B 0,C 180,E1 -6689.273,E2 -6689.273} C_VEL
LIN {X 0,Y 488.698,Z 142.611,A -85,B 0,C 180,E1 -6692.148,E2 -6692.148} C_VEL
LIN {X 0,Y 488.716,Z 142.611,A -85,B 0,C 180,E1 -6695.115,E2 -6695.115} C_VEL
LIN {X 0,Y 488.728,Z 142.611,A -85,B 0,C 180,E1 -6696.854,E2 -6696.854} C_VEL
LIN {X 0,Y 489.761,Z 148.822,A -85,B 0,C 180,E1 -6698.101,E2 -6698.101} C_VEL
LIN {X 0,Y 489.518,Z 163.162,A -85,B 0,C 180,E1 -6700.858,E2 -6700.858} C_VEL
LIN {X 0,Y 489.398,Z 168.118,A -85,B 0,C 180,E1 -6701.787,E2 -6701.787} C_VEL
LIN {X 0,Y 491.805,Z 180.723,A -85,B 0,C 180,E1 -6702.063,E2 -6702.063} C_VEL
LIN {X 0,Y 491.139,Z 275.353,A -85,B 0,C 180,E1 -6703.494,E2 -6703.494} C_VEL
LIN {X 0,Y 490.88,Z 288.606,A -85,B 0,C 180,E1 -6703.862,E2 -6703.862} C_VEL
LIN {X 0,Y 490.569,Z 301.91,A -85,B 0,C 180,E1 -6704.416,E2 -6704.416} C_VEL
LIN {X 0,Y 490.105,Z 314.554,A -85,B 0,C 180,E1 -6705.145,E2 -6705.145} C_VEL
LIN {X 0,Y 489.773,Z 325.743,A -85,B 0,C 180,E1 -6705.978,E2 -6705.978} C_VEL
LIN {X 0,Y 489.362,Z 334.72,A -85,B 0,C 180,E1 -6706.801,E2 -6706.801} C_VEL
LIN {X 0,Y 489.134,Z 340.808,A -85,B 0,C 180,E1 -6707.46,E2 -6707.46} C_VEL
LIN {X 0,Y 488.243,Z 344.994,A -85,B 0,C 180,E1 -6707.946,E2 -6707.946} C_VEL
LIN {X 0,Y 485.166,Z 351.421,A -85,B 0,C 180,E1 -6708.761,E2 -6708.761} C_VEL
LIN {X 0,Y 482.14,Z 357.231,A -85,B 0,C 180,E1 -6709.64,E2 -6709.64} C_VEL
LIN {X 0,Y 481.332,Z 360.417,A -85,B 0,C 180,E1 -6710.22,E2 -6710.22} C_VEL
LIN {X 0,Y 481.135,Z 366.772,A -85,B 0,C 180,E1 -6711.623,E2 -6711.623} C_VEL
LIN {X 0,Y 480.956,Z 372.103,A -85,B 0,C 180,E1 -6713.193,E2 -6713.193} C_VEL
LIN {X 0,Y 480.836,Z 374.709,A -85,B 0,C 180,E1 -6714.221,E2 -6714.221} C_VEL
LIN {X 0,Y 480.753,Z 376.649,A -85,B 0,C 180,E1 -6715.24,E2 -6715.24} C_VEL
LIN {X 0,Y 480.703,Z 378.134,A -85,B 0,C 180,E1 -6716.445,E2 -6716.445} C_VEL
LIN {X 0,Y 480.71,Z 378.863,A -85,B 0,C 180,E1 -6717.991,E2 -6717.991} C_VEL
LIN {X 0,Y 480.763,Z 378.152,A -85,B 0,C 180,E1 -6719.597,E2 -6719.597} C_VEL
LIN {X 0,Y 480.824,Z 375.852,A -85,B 0,C 180,E1 -6721.282,E2 -6721.282} C_VEL
LIN {X 0,Y 480.929,Z 372.885,A -85,B 0,C 180,E1 -6722.592,E2 -6722.592} C_VEL
LIN {X 0,Y 481.109,Z 368.43,A -85,B 0,C 180,E1 -6724.008,E2 -6724.008} C_VEL
LIN {X 0,Y 481.256,Z 362.586,A -85,B 0,C 180,E1 -6725.405,E2 -6725.405} C_VEL
LIN {X 0,Y 481.534,Z 355.18,A -85,B 0,C 180,E1 -6726.792,E2 -6726.792} C_VEL
LIN {X 0,Y 481.848,Z 347.553,A -85,B 0,C 180,E1 -6727.94,E2 -6727.94} C_VEL
LIN {X 0,Y 482.258,Z 337.447,A -85,B 0,C 180,E1 -6729.161,E2 -6729.161} C_VEL
LIN {X 0,Y 482.654,Z 327.844,A -85,B 0,C 180,E1 -6730.101,E2 -6730.101} C_VEL
LIN {X 0,Y 483.176,Z 316.545,A -85,B 0,C 180,E1 -6730.989,E2 -6730.989} C_VEL
LIN {X 0,Y 483.561,Z 304.286,A -85,B 0,C 180,E1 -6731.736,E2 -6731.736} C_VEL
LIN {X 0,Y 483.892,Z 292.08,A -85,B 0,C 180,E1 -6732.296,E2 -6732.296} C_VEL
LIN {X 0,Y 484.16,Z 279.935,A -85,B 0,C 180,E1 -6732.688,E2 -6732.688} C_VEL
LIN {X 0,Y 484.332,Z 265.286,A -85,B 0,C 180,E1 -6732.966,E2 -6732.966} C_VEL
LIN {X 0,Y 484.891,Z 181.351,A -85,B 0,C 180,E1 -6734.234,E2 -6734.234} C_VEL
LIN {X 0,Y 482.385,Z 168.058,A -85,B 0,C 180,E1 -6734.536,E2 -6734.536} C_VEL
LIN {X 0,Y 482.896,Z 151.637,A -85,B 0,C 180,E1 -6737.817,E2 -6737.817} C_VEL
LIN {X 0,Y 482.472,Z 147.586,A -85,B 0,C 180,E1 -6738.659,E2 -6738.659} C_VEL
LIN {X 0,Y 481.735,Z 143.479,A -85,B 0,C 180,E1 -6739.546,E2 -6739.546} C_VEL
LIN {X 0,Y 481.761,Z 143.477,A -85,B 0,C 180,E1 -6742.747,E2 -6742.747} C_VEL
LIN {X 0,Y 481.771,Z 143.471,A -85,B 0,C 180,E1 -6744.979,E2 -6744.979} C_VEL
LIN {X 0,Y 481.921,Z 143.45,A -85,B 0,C 180,E1 -6747.492,E2 -6747.492} C_VEL
LIN {X 0,Y 481.917,Z 143.454,A -85,B 0,C 180,E1 -6750,E2 -6750} C_VEL
LIN {X 0,Y 481.912,Z 143.457,A -85,B 0,C 180,E1 -6752.508,E2 -6752.508} C_VEL
LIN {X 0,Y 481.779,Z 143.471,A -85,B 0,C 180,E1 -6755.861,E2 -6755.861} C_VEL
LIN {X 0,Y 481.725,Z 143.48,A -85,B 0,C 180,E1 -6758.389,E2 -6758.389} C_VEL
LIN {X 0,Y 481.754,Z 143.475,A -85,B 0,C 180,E1 -6761.785,E2 -6761.785} C_VEL
LIN {X 0,Y 481.733,Z 143.474,A -85,B 0,C 180,E1 -6765.225,E2 -6765.225} C_VEL
LIN {X 0,Y 481.707,Z 143.477,A -85,B 0,C 180,E1 -6768.722,E2 -6768.722} C_VEL
LIN {X 0,Y 481.647,Z 143.487,A -85,B 0,C 180,E1 -6771.395,E2 -6771.395} C_VEL
LIN {X 0,Y 481.651,Z 143.488,A -85,B 0,C 180,E1 -6774.115,E2 -6774.115} C_VEL
LIN {X 0,Y 481.656,Z 143.485,A -85,B 0,C 180,E1 -6777.117,E2 -6777.117} C_VEL
LIN {X 0,Y 481.669,Z 143.489,A -85,B 0,C 180,E1 -6779.742,E2 -6779.742} C_VEL
LIN {X 0,Y 481.655,Z 143.483,A -85,B 0,C 180,E1 -6782.676,E2 -6782.676} C_VEL
LIN {X 0,Y 481.633,Z 143.492,A -85,B 0,C 180,E1 -6785.71,E2 -6785.71} C_VEL
LIN {X 0,Y 481.669,Z 143.483,A -85,B 0,C 180,E1 -6788.86,E2 -6788.86} C_VEL
LIN {X 0,Y 481.618,Z 143.488,A -85,B 0,C 180,E1 -6792.164,E2 -6792.164} C_VEL
LIN {X 0,Y 481.657,Z 143.483,A -85,B 0,C 180,E1 -6794.458,E2 -6794.458} C_VEL
LIN {X 0,Y 481.618,Z 143.491,A -85,B 0,C 180,E1 -6796.855,E2 -6796.855} C_VEL
LIN {X 0,Y 481.66,Z 143.483,A -85,B 0,C 180,E1 -6800.058,E2 -6800.058} C_VEL
LIN {X 0,Y 481.623,Z 143.493,A -85,B 0,C 180,E1 -6803.253,E2 -6803.253} C_VEL
LIN {X 0,Y 481.674,Z 143.482,A -85,B 0,C 180,E1 -6806.327,E2 -6806.327} C_VEL
LIN {X 0,Y 481.637,Z 143.488,A -85,B 0,C 180,E1 -6809.421,E2 -6809.421} C_VEL
LIN {X 0,Y 481.653,Z 143.484,A -85,B 0,C 180,E1 -6812.165,E2 -6812.165} C_VEL
LIN {X 0,Y 481.677,Z 143.487,A -85,B 0,C 180,E1 -6814.967,E2 -6814.967} C_VEL
LIN {X 0,Y 481.64,Z 143.485,A -85,B 0,C 180,E1 -6817.704,E2 -6817.704} C_VEL
LIN {X 0,Y 481.697,Z 143.483,A -85,B 0,C 180,E1 -6820.393,E2 -6820.393} C_VEL
LIN {X 0,Y 481.618,Z 143.491,A -85,B 0,C 180,E1 -6823.031,E2 -6823.031} C_VEL
LIN {X 0,Y 481.67,Z 143.482,A -85,B 0,C 180,E1 -6825.638,E2 -6825.638} C_VEL
LIN {X 0,Y 481.756,Z 143.475,A -85,B 0,C 180,E1 -6828.215,E2 -6828.215} C_VEL
LIN {X 0,Y 481.721,Z 143.475,A -85,B 0,C 180,E1 -6831.611,E2 -6831.611} C_VEL
LIN {X 0,Y 481.777,Z 143.474,A -85,B 0,C 180,E1 -6834.139,E2 -6834.139} C_VEL
LIN {X 0,Y 481.911,Z 143.452,A -85,B 0,C 180,E1 -6837.492,E2 -6837.492} C_VEL
LIN {X 0,Y 481.914,Z 143.457,A -85,B 0,C 180,E1 -6840,E2 -6840} C_VEL
LIN {X 0,Y 481.91,Z 143.455,A -85,B 0,C 180,E1 -6842.508,E2 -6842.508} C_VEL
LIN {X 0,Y 481.775,Z 143.474,A -85,B 0,C 180,E1 -6845.861,E2 -6845.861} C_VEL
LIN {X 0,Y 481.72,Z 143.478,A -85,B 0,C 180,E1 -6848.389,E2 -6848.389} C_VEL
LIN {X 0,Y 481.739,Z 143.48,A -85,B 0,C 180,E1 -6851.785,E2 -6851.785} C_VEL
LIN {X 0,Y 481.696,Z 143.48,A -85,B 0,C 180,E1 -6855.226,E2 -6855.226} C_VEL
LIN {X 0,Y 481.643,Z 143.485,A -85,B 0,C 180,E1 -6858.725,E2 -6858.725} C_VEL
LIN {X 0,Y 481.624,Z 143.492,A -85,B 0,C 180,E1 -6861.396,E2 -6861.396} C_VEL
LIN {X 0,Y 481.644,Z 143.487,A -85,B 0,C 180,E1 -6864.115,E2 -6864.115} C_VEL
LIN {X 0,Y 481.645,Z 143.488,A -85,B 0,C 180,E1 -6867.114,E2 -6867.114} C_VEL
LIN {X 0,Y 481.603,Z 143.494,A -85,B 0,C 180,E1 -6869.746,E2 -6869.746} C_VEL
LIN {X 0,Y 481.636,Z 143.486,A -85,B 0,C 180,E1 -6872.677,E2 -6872.677} C_VEL
LIN {X 0,Y 481.65,Z 143.49,A -85,B 0,C 180,E1 -6875.201,E2 -6875.201} C_VEL
LIN {X 0,Y 481.628,Z 143.487,A -85,B 0,C 180,E1 -6878.003,E2 -6878.003} C_VEL
LIN {X 0,Y 481.624,Z 143.493,A -85,B 0,C 180,E1 -6881.045,E2 -6881.045} C_VEL
LIN {X 0,Y 481.652,Z 143.485,A -85,B 0,C 180,E1 -6884.458,E2 -6884.458} C_VEL
LIN {X 0,Y 481.614,Z 143.494,A -85,B 0,C 180,E1 -6886.856,E2 -6886.856} C_VEL
LIN {X 0,Y 481.631,Z 143.486,A -85,B 0,C 180,E1 -6890.055,E2 -6890.055} C_VEL
LIN {X 0,Y 481.605,Z 143.493,A -85,B 0,C 180,E1 -6893.251,E2 -6893.251} C_VEL
LIN {X 0,Y 481.672,Z 143.483,A -85,B 0,C 180,E1 -6896.327,E2 -6896.327} C_VEL
LIN {X 0,Y 481.612,Z 143.492,A -85,B 0,C 180,E1 -6899.426,E2 -6899.426} C_VEL
LIN {X 0,Y 481.643,Z 143.489,A -85,B 0,C 180,E1 -6902.164,E2 -6902.164} C_VEL
LIN {X 0,Y 481.646,Z 143.515,A -85,B 0,C 180,E1 -6904.781,E2 -6904.781} C_VEL
LIN {X 0,Y 483.497,Z 153.33,A -85,B 0,C 180,E1 -6906.638,E2 -6906.638} C_VEL
LIN {X 0,Y 483.4,Z 162.323,A -85,B 0,C 180,E1 -6908.23,E2 -6908.23} C_VEL
LIN {X 0,Y 482.721,Z 180.117,A -85,B 0,C 180,E1 -6911.319,E2 -6911.319} C_VEL
LIN {X 0,Y 482.267,Z 192.809,A -85,B 0,C 180,E1 -6913.497,E2 -6913.497} C_VEL
LIN {X 0,Y 484.832,Z 209.789,A -85,B 0,C 180,E1 -6913.849,E2 -6913.849} C_VEL
LIN {X 0,Y 484.139,Z 301.655,A -85,B 0,C 180,E1 -6915.256,E2 -6915.256} C_VEL
LIN {X 0,Y 483.857,Z 315.421,A -85,B 0,C 180,E1 -6915.651,E2 -6915.651} C_VEL
LIN {X 0,Y 483.415,Z 327.795,A -85,B 0,C 180,E1 -6916.174,E2 -6916.174} C_VEL
LIN {X 0,Y 483.005,Z 339.669,A -85,B 0,C 180,E1 -6916.859,E2 -6916.859} C_VEL
LIN {X 0,Y 482.544,Z 351.212,A -85,B 0,C 180,E1 -6917.712,E2 -6917.712} C_VEL
LIN {X 0,Y 482.177,Z 361.385,A -85,B 0,C 180,E1 -6918.652,E2 -6918.652} C_VEL
LIN {X 0,Y 481.719,Z 370.629,A -85,B 0,C 180,E1 -6919.705,E2 -6919.705} C_VEL
LIN {X 0,Y 481.384,Z 379.622,A -85,B 0,C 180,E1 -6920.97,E2 -6920.97} C_VEL
LIN {X 0,Y 481.134,Z 386.863,A -85,B 0,C 180,E1 -6922.235,E2 -6922.235} C_VEL
LIN {X 0,Y 480.944,Z 392.871,A -85,B 0,C 180,E1 -6923.556,E2 -6923.556} C_VEL
LIN {X 0,Y 480.894,Z 397.817,A -85,B 0,C 180,E1 -6924.969,E2 -6924.969} C_VEL
LIN {X 0,Y 480.826,Z 400.12,A -85,B 0,C 180,E1 -6925.809,E2 -6925.809} C_VEL
LIN {X 0,Y 480.888,Z 401.993,A -85,B 0,C 180,E1 -6926.649,E2 -6926.649} C_VEL
LIN {X 0,Y 480.823,Z 403.393,A -85,B 0,C 180,E1 -6927.487,E2 -6927.487} C_VEL
LIN {X 0,Y 480.792,Z 404.391,A -85,B 0,C 180,E1 -6928.325,E2 -6928.325} C_VEL
LIN {X 0,Y 480.761,Z 404.998,A -85,B 0,C 180,E1 -6929.162,E2 -6929.162} C_VEL
LIN {X 0,Y 480.746,Z 405.212,A -85,B 0,C 180,E1 -6930,E2 -6930} C_VEL
LIN {X 0,Y 480.761,Z 404.993,A -85,B 0,C 180,E1 -6930.838,E2 -6930.838} C_VEL
LIN {X 0,Y 480.792,Z 404.379,A -85,B 0,C 180,E1 -6931.675,E2 -6931.675} C_VEL
LIN {X 0,Y 480.823,Z 403.377,A -85,B 0,C 180,E1 -6932.513,E2 -6932.513} C_VEL
LIN {X 0,Y 480.888,Z 401.972,A -85,B 0,C 180,E1 -6933.351,E2 -6933.351} C_VEL
LIN {X 0,Y 480.837,Z 399.015,A -85,B 0,C 180,E1 -6934.611,E2 -6934.611} C_VEL
LIN {X 0,Y 480.917,Z 395.018,A -85,B 0,C 180,E1 -6935.871,E2 -6935.871} C_VEL
LIN {X 0,Y 481.104,Z 388.87,A -85,B 0,C 180,E1 -6937.344,E2 -6937.344} C_VEL
LIN {X 0,Y 481.304,Z 382.154,A -85,B 0,C 180,E1 -6938.608,E2 -6938.608} C_VEL
LIN {X 0,Y 481.622,Z 373.824,A -85,B 0,C 180,E1 -6939.873,E2 -6939.873} C_VEL
LIN {X 0,Y 481.985,Z 365.274,A -85,B 0,C 180,E1 -6940.927,E2 -6940.927} C_VEL
LIN {X 0,Y 482.438,Z 354.742,A -85,B 0,C 180,E1 -6941.979,E2 -6941.979} C_VEL
LIN {X 0,Y 482.865,Z 343.34,A -85,B 0,C 180,E1 -6942.894,E2 -6942.894} C_VEL
LIN {X 0,Y 483.227,Z 332.803,A -85,B 0,C 180,E1 -6943.563,E2 -6943.563} C_VEL
LIN {X 0,Y 483.632,Z 320.961,A -85,B 0,C 180,E1 -6944.141,E2 -6944.141} C_VEL
LIN {X 0,Y 484.036,Z 307.316,A -85,B 0,C 180,E1 -6944.612,E2 -6944.612} C_VEL
LIN {X 0,Y 484.314,Z 293.415,A -85,B 0,C 180,E1 -6944.899,E2 -6944.899} C_VEL
LIN {X 0,Y 484.81,Z 208.866,A -85,B 0,C 180,E1 -6946.18,E2 -6946.18} C_VEL
LIN {X 0,Y 482.246,Z 192.397,A -85,B 0,C 180,E1 -6946.54,E2 -6946.54} C_VEL
LIN {X 0,Y 482.8,Z 175.908,A -85,B 0,C 180,E1 -6949.351,E2 -6949.351} C_VEL
LIN {X 0,Y 483.398,Z 159.356,A -85,B 0,C 180,E1 -6952.211,E2 -6952.211} C_VEL
LIN {X 0,Y 483.563,Z 154.234,A -85,B 0,C 180,E1 -6953.105,E2 -6953.105} C_VEL
LIN {X 0,Y 481.662,Z 143.49,A -85,B 0,C 180,E1 -6955.128,E2 -6955.128} C_VEL
LIN {X 0,Y 481.643,Z 143.492,A -85,B 0,C 180,E1 -6957.836,E2 -6957.836} C_VEL
LIN {X 0,Y 481.61,Z 143.496,A -85,B 0,C 180,E1 -6960.714,E2 -6960.714} C_VEL
LIN {X 0,Y 481.651,Z 143.489,A -85,B 0,C 180,E1 -6963.724,E2 -6963.724} C_VEL
LIN {X 0,Y 481.601,Z 143.494,A -85,B 0,C 180,E1 -6966.75,E2 -6966.75} C_VEL
LIN {X 0,Y 481.629,Z 143.489,A -85,B 0,C 180,E1 -6969.946,E2 -6969.946} C_VEL
LIN {X 0,Y 481.616,Z 143.495,A -85,B 0,C 180,E1 -6973.303,E2 -6973.303} C_VEL
LIN {X 0,Y 481.65,Z 143.487,A -85,B 0,C 180,E1 -6975.642,E2 -6975.642} C_VEL
LIN {X 0,Y 481.606,Z 143.497,A -85,B 0,C 180,E1 -6978.953,E2 -6978.953} C_VEL
LIN {X 0,Y 481.623,Z 143.488,A -85,B 0,C 180,E1 -6981.998,E2 -6981.998} C_VEL
LIN {X 0,Y 481.671,Z 143.484,A -85,B 0,C 180,E1 -6985.316,E2 -6985.316} C_VEL
LIN {X 0,Y 481.622,Z 143.489,A -85,B 0,C 180,E1 -6988.31,E2 -6988.31} C_VEL
LIN {X 0,Y 481.636,Z 143.486,A -85,B 0,C 180,E1 -6991.214,E2 -6991.214} C_VEL
LIN {X 0,Y 481.621,Z 143.489,A -85,B 0,C 180,E1 -6994.038,E2 -6994.038} C_VEL
LIN {X 0,Y 481.637,Z 143.491,A -85,B 0,C 180,E1 -6996.824,E2 -6996.824} C_VEL
LIN {X 0,Y 481.621,Z 143.483,A -85,B 0,C 180,E1 -6999.499,E2 -6999.499} C_VEL
LIN {X 0,Y 481.649,Z 143.488,A -85,B 0,C 180,E1 -7002.156,E2 -7002.156} C_VEL
LIN {X 0,Y 481.694,Z 143.482,A -85,B 0,C 180,E1 -7004.774,E2 -7004.774} C_VEL
LIN {X 0,Y 481.73,Z 143.479,A -85,B 0,C 180,E1 -7008.215,E2 -7008.215} C_VEL
LIN {X 0,Y 481.716,Z 143.476,A -85,B 0,C 180,E1 -7011.611,E2 -7011.611} C_VEL
LIN {X 0,Y 481.768,Z 143.47,A -85,B 0,C 180,E1 -7014.139,E2 -7014.139} C_VEL
LIN {X 0,Y 481.909,Z 143.45,A -85,B 0,C 180,E1 -7017.492,E2 -7017.492} C_VEL
LIN {X 0,Y 481.914,Z 143.457,A -85,B 0,C 180,E1 -7020,E2 -7020} C_VEL
LIN {X 0,Y 481.91,Z 143.454,A -85,B 0,C 180,E1 -7022.508,E2 -7022.508} C_VEL
LIN {X 0,Y 481.776,Z 143.472,A -85,B 0,C 180,E1 -7025.861,E2 -7025.861} C_VEL
LIN {X 0,Y 481.72,Z 143.477,A -85,B 0,C 180,E1 -7028.389,E2 -7028.389} C_VEL
LIN {X 0,Y 481.74,Z 143.481,A -85,B 0,C 180,E1 -7031.785,E2 -7031.785} C_VEL
LIN {X 0,Y 481.733,Z 143.476,A -85,B 0,C 180,E1 -7035.225,E2 -7035.225} C_VEL
LIN {X 0,Y 481.653,Z 143.484,A -85,B 0,C 180,E1 -7038.724,E2 -7038.724} C_VEL
LIN {X 0,Y 481.633,Z 143.49,A -85,B 0,C 180,E1 -7041.395,E2 -7041.395} C_VEL
LIN {X 0,Y 481.65,Z 143.489,A -85,B 0,C 180,E1 -7044.115,E2 -7044.115} C_VEL
LIN {X 0,Y 481.655,Z 143.489,A -85,B 0,C 180,E1 -7047.117,E2 -7047.117} C_VEL
LIN {X 0,Y 481.657,Z 143.49,A -85,B 0,C 180,E1 -7049.743,E2 -7049.743} C_VEL
LIN {X 0,Y 481.655,Z 143.487,A -85,B 0,C 180,E1 -7052.676,E2 -7052.676} C_VEL
LIN {X 0,Y 481.642,Z 143.494,A -85,B 0,C 180,E1 -7055.709,E2 -7055.709} C_VEL
LIN {X 0,Y 481.705,Z 143.559,A -85,B 0,C 180,E1 -7056.694,E2 -7056.694} C_VEL
LIN {X 0,Y 482.838,Z 150.884,A -85,B 0,C 180,E1 -7058.186,E2 -7058.186} C_VEL
LIN {X 0,Y 482.51,Z 165.173,A -85,B 0,C 180,E1 -7060.954,E2 -7060.954} C_VEL
LIN {X 0,Y 482.411,Z 168.183,A -85,B 0,C 180,E1 -7061.537,E2 -7061.537} C_VEL
LIN {X 0,Y 485.038,Z 182.26,A -85,B 0,C 180,E1 -7061.852,E2 -7061.852} C_VEL
LIN {X 0,Y 484.273,Z 275.816,A -85,B 0,C 180,E1 -7063.288,E2 -7063.288} C_VEL
LIN {X 0,Y 484.021,Z 289.329,A -85,B 0,C 180,E1 -7063.674,E2 -7063.674} C_VEL
LIN {X 0,Y 483.691,Z 302.191,A -85,B 0,C 180,E1 -7064.222,E2 -7064.222} C_VEL
LIN {X 0,Y 483.195,Z 314.531,A -85,B 0,C 180,E1 -7064.941,E2 -7064.941} C_VEL
LIN {X 0,Y 482.83,Z 326.21,A -85,B 0,C 180,E1 -7065.824,E2 -7065.824} C_VEL
LIN {X 0,Y 482.374,Z 336.302,A -85,B 0,C 180,E1 -7066.782,E2 -7066.782} C_VEL
LIN {X 0,Y 481.957,Z 345.609,A -85,B 0,C 180,E1 -7067.872,E2 -7067.872} C_VEL
LIN {X 0,Y 481.628,Z 353.197,A -85,B 0,C 180,E1 -7068.955,E2 -7068.955} C_VEL
LIN {X 0,Y 481.332,Z 360.417,A -85,B 0,C 180,E1 -7070.22,E2 -7070.22} C_VEL
LIN {X 0,Y 480.52,Z 363.419,A -85,B 0,C 180,E1 -7070.82,E2 -7070.82} C_VEL
LIN {X 0,Y 477.505,Z 367.808,A -85,B 0,C 180,E1 -7071.82,E2 -7071.82} C_VEL
LIN {X 0,Y 474.542,Z 371.555,A -85,B 0,C 180,E1 -7072.871,E2 -7072.871} C_VEL
LIN {X 0,Y 473.822,Z 373.431,A -85,B 0,C 180,E1 -7073.543,E2 -7073.543} C_VEL
LIN {X 0,Y 473.706,Z 375.98,A -85,B 0,C 180,E1 -7074.686,E2 -7074.686} C_VEL
LIN {X 0,Y 473.63,Z 378.123,A -85,B 0,C 180,E1 -7076.198,E2 -7076.198} C_VEL
LIN {X 0,Y 473.614,Z 379.017,A -85,B 0,C 180,E1 -7077.761,E2 -7077.761} C_VEL
LIN {X 0,Y 473.651,Z 378.555,A -85,B 0,C 180,E1 -7079.384,E2 -7079.384} C_VEL
LIN {X 0,Y 473.726,Z 376.465,A -85,B 0,C 180,E1 -7081.081,E2 -7081.081} C_VEL
LIN {X 0,Y 473.862,Z 373.149,A -85,B 0,C 180,E1 -7082.627,E2 -7082.627} C_VEL
LIN {X 0,Y 474.055,Z 368.723,A -85,B 0,C 180,E1 -7084.065,E2 -7084.065} C_VEL
LIN {X 0,Y 474.187,Z 362.914,A -85,B 0,C 180,E1 -7085.481,E2 -7085.481} C_VEL
LIN {X 0,Y 474.439,Z 356.637,A -85,B 0,C 180,E1 -7086.697,E2 -7086.697} C_VEL
LIN {X 0,Y 474.831,Z 347.934,A -85,B 0,C 180,E1 -7088.054,E2 -7088.054} C_VEL
LIN {X 0,Y 475.244,Z 338.62,A -85,B 0,C 180,E1 -7089.211,E2 -7089.211} C_VEL
LIN {X 0,Y 475.679,Z 328.402,A -85,B 0,C 180,E1 -7090.239,E2 -7090.239} C_VEL
LIN {X 0,Y 476.153,Z 318.411,A -85,B 0,C 180,E1 -7091.051,E2 -7091.051} C_VEL
LIN {X 0,Y 476.552,Z 307.974,A -85,B 0,C 180,E1 -7091.736,E2 -7091.736} C_VEL
LIN {X 0,Y 476.905,Z 295.631,A -85,B 0,C 180,E1 -7092.361,E2 -7092.361} C_VEL
LIN {X 0,Y 477.216,Z 282.965,A -85,B 0,C 180,E1 -7092.815,E2 -7092.815} C_VEL
LIN {X 0,Y 477.446,Z 269.692,A -85,B 0,C 180,E1 -7093.113,E2 -7093.113} C_VEL
LIN {X 0,Y 478.108,Z 182.385,A -85,B 0,C 180,E1 -7094.45,E2 -7094.45} C_VEL
LIN {X 0,Y 475.419,Z 168.184,A -85,B 0,C 180,E1 -7094.788,E2 -7094.788} C_VEL
LIN {X 0,Y 475.927,Z 153.027,A -85,B 0,C 180,E1 -7097.852,E2 -7097.852} C_VEL
LIN {X 0,Y 475.379,Z 147.968,A -85,B 0,C 180,E1 -7098.919,E2 -7098.919} C_VEL
LIN {X 0,Y 474.674,Z 144.359,A -85,B 0,C 180,E1 -7099.712,E2 -7099.712} C_VEL
LIN {X 0,Y 474.717,Z 144.354,A -85,B 0,C 180,E1 -7102.708,E2 -7102.708} C_VEL
LIN {X 0,Y 474.742,Z 144.348,A -85,B 0,C 180,E1 -7104.904,E2 -7104.904} C_VEL
LIN {X 0,Y 474.887,Z 144.326,A -85,B 0,C 180,E1 -7107.455,E2 -7107.455} C_VEL
LIN {X 0,Y 474.886,Z 144.33,A -85,B 0,C 180,E1 -7110,E2 -7110} C_VEL
LIN {X 0,Y 474.877,Z 144.333,A -85,B 0,C 180,E1 -7112.545,E2 -7112.545} C_VEL
LIN {X 0,Y 474.741,Z 144.349,A -85,B 0,C 180,E1 -7115.948,E2 -7115.948} C_VEL
LIN {X 0,Y 474.7,Z 144.353,A -85,B 0,C 180,E1 -7118.514,E2 -7118.514} C_VEL
LIN {X 0,Y 474.708,Z 144.355,A -85,B 0,C 180,E1 -7121.962,E2 -7121.962} C_VEL
LIN {X 0,Y 474.691,Z 144.353,A -85,B 0,C 180,E1 -7125.456,E2 -7125.456} C_VEL
LIN {X 0,Y 474.661,Z 144.355,A -85,B 0,C 180,E1 -7129.011,E2 -7129.011} C_VEL
LIN {X 0,Y 474.59,Z 144.37,A -85,B 0,C 180,E1 -7131.729,E2 -7131.729} C_VEL
LIN {X 0,Y 474.629,Z 144.359,A -85,B 0,C 180,E1 -7134.495,E2 -7134.495} C_VEL
LIN {X 0,Y 474.602,Z 144.365,A -85,B 0,C 180,E1 -7137.326,E2 -7137.326} C_VEL
LIN {X 0,Y 474.6,Z 144.364,A -85,B 0,C 180,E1 -7140.231,E2 -7140.231} C_VEL
LIN {X 0,Y 474.617,Z 144.364,A -85,B 0,C 180,E1 -7143.222,E2 -7143.222} C_VEL
LIN {X 0,Y 474.586,Z 144.364,A -85,B 0,C 180,E1 -7146.324,E2 -7146.324} C_VEL
LIN {X 0,Y 474.625,Z 144.365,A -85,B 0,C 180,E1 -7149.548,E2 -7149.548} C_VEL
LIN {X 0,Y 474.579,Z 144.365,A -85,B 0,C 180,E1 -7152.23,E2 -7152.23} C_VEL
LIN {X 0,Y 474.619,Z 144.368,A -85,B 0,C 180,E1 -7155.298,E2 -7155.298} C_VEL
LIN {X 0,Y 474.595,Z 144.363,A -85,B 0,C 180,E1 -7158.212,E2 -7158.212} C_VEL
LIN {X 0,Y 474.611,Z 144.364,A -85,B 0,C 180,E1 -7161.542,E2 -7161.542} C_VEL
LIN {X 0,Y 474.623,Z 144.363,A -85,B 0,C 180,E1 -7164.725,E2 -7164.725} C_VEL
LIN {X 0,Y 474.629,Z 144.359,A -85,B 0,C 180,E1 -7167.787,E2 -7167.787} C_VEL
LIN {X 0,Y 474.597,Z 144.371,A -85,B 0,C 180,E1 -7170.891,E2 -7170.891} C_VEL
LIN {X 0,Y 474.594,Z 144.363,A -85,B 0,C 180,E1 -7173.624,E2 -7173.624} C_VEL
LIN {X 0,Y 474.637,Z 144.364,A -85,B 0,C 180,E1 -7176.642,E2 -7176.642} C_VEL
LIN {X 0,Y 474.646,Z 144.358,A -85,B 0,C 180,E1 -7180.089,E2 -7180.089} C_VEL
LIN {X 0,Y 474.593,Z 144.369,A -85,B 0,C 180,E1 -7182.772,E2 -7182.772} C_VEL
LIN {X 0,Y 474.63,Z 144.358,A -85,B 0,C 180,E1 -7185.42,E2 -7185.42} C_VEL
LIN {X 0,Y 474.709,Z 144.351,A -85,B 0,C 180,E1 -7188.038,E2 -7188.038} C_VEL
LIN {X 0,Y 474.67,Z 144.353,A -85,B 0,C 180,E1 -7191.485,E2 -7191.485} C_VEL
LIN {X 0,Y 474.74,Z 144.349,A -85,B 0,C 180,E1 -7194.052,E2 -7194.052} C_VEL
LIN {X 0,Y 474.876,Z 144.328,A -85,B 0,C 180,E1 -7197.455,E2 -7197.455} C_VEL
LIN {X 0,Y 474.884,Z 144.332,A -85,B 0,C 180,E1 -7200,E2 -7200} C_VEL
LIN {X 0,Y 474.875,Z 144.331,A -85,B 0,C 180,E1 -7202.545,E2 -7202.545} C_VEL
LIN {X 0,Y 474.739,Z 144.352,A -85,B 0,C 180,E1 -7205.948,E2 -7205.948} C_VEL
LIN {X 0,Y 474.668,Z 144.355,A -85,B 0,C 180,E1 -7208.515,E2 -7208.515} C_VEL
LIN {X 0,Y 474.697,Z 144.358,A -85,B 0,C 180,E1 -7211.963,E2 -7211.963} C_VEL
LIN {X 0,Y 474.654,Z 144.359,A -85,B 0,C 180,E1 -7215.457,E2 -7215.457} C_VEL
LIN {X 0,Y 474.596,Z 144.363,A -85,B 0,C 180,E1 -7219.013,E2 -7219.013} C_VEL
LIN {X 0,Y 474.573,Z 144.373,A -85,B 0,C 180,E1 -7221.73,E2 -7221.73} C_VEL
LIN {X 0,Y 474.623,Z 144.359,A -85,B 0,C 180,E1 -7224.495,E2 -7224.495} C_VEL
LIN {X 0,Y 474.595,Z 144.368,A -85,B 0,C 180,E1 -7227.327,E2 -7227.327} C_VEL
LIN {X 0,Y 474.552,Z 144.368,A -85,B 0,C 180,E1 -7230.234,E2 -7230.234} C_VEL
LIN {X 0,Y 474.61,Z 144.367,A -85,B 0,C 180,E1 -7233.223,E2 -7233.223} C_VEL
LIN {X 0,Y 474.571,Z 144.366,A -85,B 0,C 180,E1 -7236.325,E2 -7236.325} C_VEL
LIN {X 0,Y 474.605,Z 144.365,A -85,B 0,C 180,E1 -7239.55,E2 -7239.55} C_VEL
LIN {X 0,Y 474.577,Z 144.365,A -85,B 0,C 180,E1 -7242.23,E2 -7242.23} C_VEL
LIN {X 0,Y 474.615,Z 144.366,A -85,B 0,C 180,E1 -7245.298,E2 -7245.298} C_VEL
LIN {X 0,Y 474.591,Z 144.364,A -85,B 0,C 180,E1 -7248.211,E2 -7248.211} C_VEL
LIN {X 0,Y 474.587,Z 144.365,A -85,B 0,C 180,E1 -7251.54,E2 -7251.54} C_VEL
LIN {X 0,Y 474.605,Z 144.368,A -85,B 0,C 180,E1 -7254.724,E2 -7254.724} C_VEL
LIN {X 0,Y 474.611,Z 144.361,A -85,B 0,C 180,E1 -7257.786,E2 -7257.786} C_VEL
LIN {X 0,Y 474.577,Z 144.373,A -85,B 0,C 180,E1 -7260.895,E2 -7260.895} C_VEL
LIN {X 0,Y 474.573,Z 144.371,A -85,B 0,C 180,E1 -7263.623,E2 -7263.623} C_VEL
LIN {X 0,Y 474.603,Z 144.458,A -85,B 0,C 180,E1 -7264.595,E2 -7264.595} C_VEL
LIN {X 0,Y 476.543,Z 154.544,A -85,B 0,C 180,E1 -7266.535,E2 -7266.535} C_VEL
LIN {X 0,Y 476.455,Z 162.415,A -85,B 0,C 180,E1 -7267.951,E2 -7267.951} C_VEL
LIN {X 0,Y 475.712,Z 181.168,A -85,B 0,C 180,E1 -7271.257,E2 -7271.257} C_VEL
LIN {X 0,Y 475.294,Z 192.673,A -85,B 0,C 180,E1 -7273.258,E2 -7273.258} C_VEL
LIN {X 0,Y 478.005,Z 210.7,A -85,B 0,C 180,E1 -7273.634,E2 -7273.634} C_VEL
LIN {X 0,Y 477.278,Z 301.168,A -85,B 0,C 180,E1 -7275.04,E2 -7275.04} C_VEL
LIN {X 0,Y 476.992,Z 315.033,A -85,B 0,C 180,E1 -7275.44,E2 -7275.44} C_VEL
LIN {X 0,Y 476.509,Z 327.47,A -85,B 0,C 180,E1 -7275.97,E2 -7275.97} C_VEL
LIN {X 0,Y 476.044,Z 339.851,A -85,B 0,C 180,E1 -7276.696,E2 -7276.696} C_VEL
LIN {X 0,Y 475.555,Z 350.899,A -85,B 0,C 180,E1 -7277.525,E2 -7277.525} C_VEL
LIN {X 0,Y 475.151,Z 361.135,A -85,B 0,C 180,E1 -7278.482,E2 -7278.482} C_VEL
LIN {X 0,Y 474.711,Z 370.396,A -85,B 0,C 180,E1 -7279.551,E2 -7279.551} C_VEL
LIN {X 0,Y 474.341,Z 379.398,A -85,B 0,C 180,E1 -7280.835,E2 -7280.835} C_VEL
LIN {X 0,Y 474.058,Z 386.646,A -85,B 0,C 180,E1 -7282.118,E2 -7282.118} C_VEL
LIN {X 0,Y 473.868,Z 393.044,A -85,B 0,C 180,E1 -7283.56,E2 -7283.56} C_VEL
LIN {X 0,Y 473.825,Z 397.612,A -85,B 0,C 180,E1 -7284.894,E2 -7284.894} C_VEL
LIN {X 0,Y 473.733,Z 399.917,A -85,B 0,C 180,E1 -7285.746,E2 -7285.746} C_VEL
LIN {X 0,Y 473.795,Z 401.793,A -85,B 0,C 180,E1 -7286.598,E2 -7286.598} C_VEL
LIN {X 0,Y 473.741,Z 403.196,A -85,B 0,C 180,E1 -7287.449,E2 -7287.449} C_VEL
LIN {X 0,Y 473.69,Z 404.803,A -85,B 0,C 180,E1 -7289.15,E2 -7289.15} C_VEL
LIN {X 0,Y 473.672,Z 405.018,A -85,B 0,C 180,E1 -7290,E2 -7290} C_VEL
LIN {X 0,Y 473.69,Z 404.8,A -85,B 0,C 180,E1 -7290.85,E2 -7290.85} C_VEL
LIN {X 0,Y 473.741,Z 403.183,A -85,B 0,C 180,E1 -7292.551,E2 -7292.551} C_VEL
LIN {X 0,Y 473.795,Z 401.778,A -85,B 0,C 180,E1 -7293.402,E2 -7293.402} C_VEL
LIN {X 0,Y 473.76,Z 398.821,A -85,B 0,C 180,E1 -7294.68,E2 -7294.68} C_VEL
LIN {X 0,Y 473.825,Z 394.821,A -85,B 0,C 180,E1 -7295.96,E2 -7295.96} C_VEL
LIN {X 0,Y 474.013,Z 388.673,A -85,B 0,C 180,E1 -7297.454,E2 -7297.454} C_VEL
LIN {X 0,Y 474.263,Z 381.958,A -85,B 0,C 180,E1 -7298.737,E2 -7298.737} C_VEL
LIN {X 0,Y 474.563,Z 373.629,A -85,B 0,C 180,E1 -7300.021,E2 -7300.021} C_VEL
LIN {X 0,Y 474.988,Z 365.084,A -85,B 0,C 180,E1 -7301.09,E2 -7301.09} C_VEL
LIN {X 0,Y 475.455,Z 354.789,A -85,B 0,C 180,E1 -7302.136,E2 -7302.136} C_VEL
LIN {X 0,Y 475.86,Z 344.373,A -85,B 0,C 180,E1 -7302.995,E2 -7302.995} C_VEL
LIN {X 0,Y 476.314,Z 332.622,A -85,B 0,C 180,E1 -7303.764,E2 -7303.764} C_VEL
LIN {X 0,Y 476.761,Z 320.79,A -85,B 0,C 180,E1 -7304.35,E2 -7304.35} C_VEL
LIN {X 0,Y 477.17,Z 307.162,A -85,B 0,C 180,E1 -7304.828,E2 -7304.828} C_VEL
LIN {X 0,Y 477.475,Z 293.33,A -85,B 0,C 180,E1 -7305.118,E2 -7305.118} C_VEL
LIN {X 0,Y 477.946,Z 209.248,A -85,B 0,C 180,E1 -7306.415,E2 -7306.415} C_VEL
LIN {X 0,Y 475.288,Z 192.12,A -85,B 0,C 180,E1 -7306.808,E2 -7306.808} C_VEL
LIN {X 0,Y 475.835,Z 175.933,A -85,B 0,C 180,E1 -7309.612,E2 -7309.612} C_VEL
LIN {X 0,Y 476.472,Z 160.468,A -85,B 0,C 180,E1 -7312.322,E2 -7312.322} C_VEL
LIN {X 0,Y 476.453,Z 154.06,A -85,B 0,C 180,E1 -7313.47,E2 -7313.47} C_VEL
LIN {X 0,Y 474.61,Z 144.368,A -85,B 0,C 180,E1 -7315.345,E2 -7315.345} C_VEL
LIN {X 0,Y 474.59,Z 144.369,A -85,B 0,C 180,E1 -7318.286,E2 -7318.286} C_VEL
LIN {X 0,Y 474.575,Z 144.375,A -85,B 0,C 180,E1 -7321.22,E2 -7321.22} C_VEL
LIN {X 0,Y 474.605,Z 144.365,A -85,B 0,C 180,E1 -7324.244,E2 -7324.244} C_VEL
LIN {X 0,Y 474.534,Z 144.377,A -85,B 0,C 180,E1 -7327.389,E2 -7327.389} C_VEL
LIN {X 0,Y 474.579,Z 144.369,A -85,B 0,C 180,E1 -7329.64,E2 -7329.64} C_VEL
LIN {X 0,Y 474.567,Z 144.374,A -85,B 0,C 180,E1 -7332.94,E2 -7332.94} C_VEL
LIN {X 0,Y 474.582,Z 144.367,A -85,B 0,C 180,E1 -7335.892,E2 -7335.892} C_VEL
LIN {X 0,Y 474.582,Z 144.37,A -85,B 0,C 180,E1 -7339.048,E2 -7339.048} C_VEL
LIN {X 0,Y 474.585,Z 144.365,A -85,B 0,C 180,E1 -7341.709,E2 -7341.709} C_VEL
LIN {X 0,Y 474.605,Z 144.367,A -85,B 0,C 180,E1 -7344.724,E2 -7344.724} C_VEL
LIN {X 0,Y 474.612,Z 144.36,A -85,B 0,C 180,E1 -7347.786,E2 -7347.786} C_VEL
LIN {X 0,Y 474.578,Z 144.367,A -85,B 0,C 180,E1 -7350.896,E2 -7350.896} C_VEL
LIN {X 0,Y 474.574,Z 144.365,A -85,B 0,C 180,E1 -7353.623,E2 -7353.623} C_VEL
LIN {X 0,Y 474.599,Z 144.369,A -85,B 0,C 180,E1 -7356.653,E2 -7356.653} C_VEL
LIN {X 0,Y 474.589,Z 144.361,A -85,B 0,C 180,E1 -7360.087,E2 -7360.087} C_VEL
LIN {X 0,Y 474.586,Z 144.367,A -85,B 0,C 180,E1 -7362.772,E2 -7362.772} C_VEL
LIN {X 0,Y 474.604,Z 144.361,A -85,B 0,C 180,E1 -7365.42,E2 -7365.42} C_VEL
LIN {X 0,Y 474.689,Z 144.355,A -85,B 0,C 180,E1 -7368.037,E2 -7368.037} C_VEL
LIN {X 0,Y 474.665,Z 144.354,A -85,B 0,C 180,E1 -7371.485,E2 -7371.485} C_VEL
LIN {X 0,Y 474.732,Z 144.346,A -85,B 0,C 180,E1 -7374.052,E2 -7374.052} C_VEL
LIN {X 0,Y 474.874,Z 144.326,A -85,B 0,C 180,E1 -7377.455,E2 -7377.455} C_VEL
LIN {X 0,Y 474.883,Z 144.332,A -85,B 0,C 180,E1 -7380,E2 -7380} C_VEL
LIN {X 0,Y 474.875,Z 144.33,A -85,B 0,C 180,E1 -7382.545,E2 -7382.545} C_VEL
LIN {X 0,Y 474.739,Z 144.349,A -85,B 0,C 180,E1 -7385.948,E2 -7385.948} C_VEL
LIN {X 0,Y 474.669,Z 144.355,A -85,B 0,C 180,E1 -7388.515,E2 -7388.515} C_VEL
LIN {X 0,Y 474.697,Z 144.356,A -85,B 0,C 180,E1 -7391.963,E2 -7391.963} C_VEL
LIN {X 0,Y 474.692,Z 144.355,A -85,B 0,C 180,E1 -7395.456,E2 -7395.456} C_VEL
LIN {X 0,Y 474.607,Z 144.363,A -85,B 0,C 180,E1 -7399.013,E2 -7399.013} C_VEL
LIN {X 0,Y 474.579,Z 144.373,A -85,B 0,C 180,E1 -7401.73,E2 -7401.73} C_VEL
LIN {X 0,Y 474.629,Z 144.362,A -85,B 0,C 180,E1 -7404.495,E2 -7404.495} C_VEL
LIN {X 0,Y 474.602,Z 144.37,A -85,B 0,C 180,E1 -7407.326,E2 -7407.326} C_VEL
LIN {X 0,Y 474.588,Z 144.367,A -85,B 0,C 180,E1 -7410.232,E2 -7410.232} C_VEL
LIN {X 0,Y 474.618,Z 144.367,A -85,B 0,C 180,E1 -7413.222,E2 -7413.222} C_VEL
LIN {X 0,Y 474.636,Z 144.41,A -85,B 0,C 180,E1 -7416.496,E2 -7416.496} C_VEL
LIN {X 0,Y 475.879,Z 151.993,A -85,B 0,C 180,E1 -7418.067,E2 -7418.067} C_VEL
LIN {X 0,Y 475.552,Z 166.015,A -85,B 0,C 180,E1 -7420.82,E2 -7420.82} C_VEL
LIN {X 0,Y 475.497,Z 168.326,A -85,B 0,C 180,E1 -7421.273,E2 -7421.273} C_VEL
LIN {X 0,Y 478.243,Z 183.389,A -85,B 0,C 180,E1 -7421.624,E2 -7421.624} C_VEL
LIN {X 0,Y 477.422,Z 276.037,A -85,B 0,C 180,E1 -7423.07,E2 -7423.07} C_VEL
LIN {X 0,Y 477.161,Z 289.488,A -85,B 0,C 180,E1 -7423.46,E2 -7423.46} C_VEL
LIN {X 0,Y 476.834,Z 301.827,A -85,B 0,C 180,E1 -7423.988,E2 -7423.988} C_VEL
LIN {X 0,Y 476.334,Z 313.821,A -85,B 0,C 180,E1 -7424.685,E2 -7424.685} C_VEL
LIN {X 0,Y 475.884,Z 325.929,A -85,B 0,C 180,E1 -7425.601,E2 -7425.601} C_VEL
LIN {X 0,Y 475.403,Z 336.411,A -85,B 0,C 180,E1 -7426.603,E2 -7426.603} C_VEL
LIN {X 0,Y 474.965,Z 345.804,A -85,B 0,C 180,E1 -7427.718,E2 -7427.718} C_VEL
LIN {X 0,Y 474.596,Z 353.895,A -85,B 0,C 180,E1 -7428.897,E2 -7428.897} C_VEL
LIN {X 0,Y 474.274,Z 360.943,A -85,B 0,C 180,E1 -7430.161,E2 -7430.161} C_VEL
LIN {X 0,Y 474.069,Z 366.84,A -85,B 0,C 180,E1 -7431.49,E2 -7431.49} C_VEL
LIN {X 0,Y 473.913,Z 370.612,A -85,B 0,C 180,E1 -7432.553,E2 -7432.553} C_VEL
LIN {X 0,Y 473.822,Z 373.431,A -85,B 0,C 180,E1 -7433.543,E2 -7433.543} C_VEL
LIN {X 0,Y 473.094,Z 375.093,A -85,B 0,C 180,E1 -7434.224,E2 -7434.224} C_VEL
LIN {X 0,Y 470.131,Z 377.251,A -85,B 0,C 180,E1 -7435.344,E2 -7435.344} C_VEL
LIN {X 0,Y 467.653,Z 378.42,A -85,B 0,C 180,E1 -7436.26,E2 -7436.26} C_VEL
LIN {X 0,Y 466.594,Z 378.953,A -85,B 0,C 180,E1 -7436.974,E2 -7436.974} C_VEL
LIN {X 0,Y 466.51,Z 379.06,A -85,B 0,C 180,E1 -7437.217,E2 -7437.217} C_VEL
LIN {X 0,Y 466.506,Z 379.235,A -85,B 0,C 180,E1 -7438.178,E2 -7438.178} C_VEL
LIN {X 0,Y 466.563,Z 378.868,A -85,B 0,C 180,E1 -7439.192,E2 -7439.192} C_VEL
LIN {X 0,Y 466.626,Z 377.074,A -85,B 0,C 180,E1 -7440.875,E2 -7440.875} C_VEL
LIN {X 0,Y 466.772,Z 373.404,A -85,B 0,C 180,E1 -7442.666,E2 -7442.666} C_VEL
LIN {X 0,Y 466.979,Z 369.013,A -85,B 0,C 180,E1 -7444.122,E2 -7444.122} C_VEL
LIN {X 0,Y 467.13,Z 363.231,A -85,B 0,C 180,E1 -7445.56,E2 -7445.56} C_VEL
LIN {X 0,Y 467.437,Z 355.881,A -85,B 0,C 180,E1 -7446.988,E2 -7446.988} C_VEL
LIN {X 0,Y 467.79,Z 348.609,A -85,B 0,C 180,E1 -7448.128,E2 -7448.128} C_VEL
LIN {X 0,Y 468.264,Z 339.035,A -85,B 0,C 180,E1 -7449.347,E2 -7449.347} C_VEL
LIN {X 0,Y 468.723,Z 328.774,A -85,B 0,C 180,E1 -7450.398,E2 -7450.398} C_VEL
LIN {X 0,Y 469.309,Z 317.363,A -85,B 0,C 180,E1 -7451.331,E2 -7451.331} C_VEL
LIN {X 0,Y 469.726,Z 305.56,A -85,B 0,C 180,E1 -7452.082,E2 -7452.082} C_VEL
LIN {X 0,Y 470.101,Z 293.441,A -85,B 0,C 180,E1 -7452.665,E2 -7452.665} C_VEL
LIN {X 0,Y 470.408,Z 280.714,A -85,B 0,C 180,E1 -7453.099,E2 -7453.099} C_VEL
LIN {X 0,Y 470.618,Z 266.421,A -85,B 0,C 180,E1 -7453.384,E2 -7453.384} C_VEL
LIN {X 0,Y 471.209,Z 182.693,A -85,B 0,C 180,E1 -7454.69,E2 -7454.69} C_VEL
LIN {X 0,Y 468.46,Z 168.394,A -85,B 0,C 180,E1 -7455.029,E2 -7455.029} C_VEL
LIN {X 0,Y 468.947,Z 153.375,A -85,B 0,C 180,E1 -7458.108,E2 -7458.108} C_VEL
LIN {X 0,Y 467.645,Z 145.236,A -85,B 0,C 180,E1 -7459.884,E2 -7459.884} C_VEL
